LIN {X 0,Y 165.96,Z 258.398,A -85,B 0,C 180,E1 -25599.436,E2 -25599.436} C_VEL
LIN {X 0,Y 163.144,Z 293.793,A -85,B 0,C 180,E1 -25600.74,E2 -25600.74} C_VEL
LIN {X 0,Y 161.079,Z 307.116,A -85,B 0,C 180,E1 -25601.609,E2 -25601.609} C_VEL
LIN {X 0,Y 157.962,Z 319.785,A -85,B 0,C 180,E1 -25602.768,E2 -25602.768} C_VEL
LIN {X 0,Y 153.973,Z 332.432,A -85,B 0,C 180,E1 -25604.505,E2 -25604.505} C_VEL
LIN {X 0,Y 149.598,Z 343.686,A -85,B 0,C 180,E1 -25606.602,E2 -25606.602} C_VEL
LIN {X 0,Y 144.876,Z 353.82,A -85,B 0,C 180,E1 -25609.089,E2 -25609.089} C_VEL
LIN {X 0,Y 140.058,Z 362.957,A -85,B 0,C 180,E1 -25612.071,E2 -25612.071} C_VEL
LIN {X 0,Y 134.888,Z 371.867,A -85,B 0,C 180,E1 -25615.937,E2 -25615.937} C_VEL
LIN {X 0,Y 130.55,Z 379.04,A -85,B 0,C 180,E1 -25620.135,E2 -25620.135} C_VEL
LIN {X 0,Y 127.194,Z 383.879,A -85,B 0,C 180,E1 -25623.767,E2 -25623.767} C_VEL
LIN {X 0,Y 123.98,Z 388.585,A -85,B 0,C 180,E1 -25628.379,E2 -25628.379} C_VEL
LIN {X 0,Y 121.649,Z 392.184,A -85,B 0,C 180,E1 -25633.21,E2 -25633.21} C_VEL
LIN {X 0,Y 120.54,Z 394.04,A -85,B 0,C 180,E1 -25636.514,E2 -25636.514} C_VEL
LIN {X 0,Y 119.326,Z 396.429,A -85,B 0,C 180,E1 -25643.235,E2 -25643.235} C_VEL
LIN {X 0,Y 119.198,Z 397.039,A -85,B 0,C 180,E1 -25646.62,E2 -25646.62} C_VEL
LIN {X 0,Y 119.291,Z 397.251,A -85,B 0,C 180,E1 -25650,E2 -25650} C_VEL
LIN {X 0,Y 119.219,Z 397.022,A -85,B 0,C 180,E1 -25653.38,E2 -25653.38} C_VEL
LIN {X 0,Y 119.788,Z 395.395,A -85,B 0,C 180,E1 -25660.138,E2 -25660.138} C_VEL
LIN {X 0,Y 120.54,Z 393.984,A -85,B 0,C 180,E1 -25663.487,E2 -25663.487} C_VEL
LIN {X 0,Y 122.284,Z 391.031,A -85,B 0,C 180,E1 -25668.427,E2 -25668.427} C_VEL
LIN {X 0,Y 124.982,Z 387.046,A -85,B 0,C 180,E1 -25673.18,E2 -25673.18} C_VEL
LIN {X 0,Y 129.119,Z 380.92,A -85,B 0,C 180,E1 -25678.442,E2 -25678.442} C_VEL
LIN {X 0,Y 130.23,Z 379.284,A -85,B 0,C 180,E1 -25679.585,E2 -25679.585} C_VEL
LIN {X 0,Y 131.603,Z 376.213,A -85,B 0,C 180,E1 -25681.706,E2 -25681.706} C_VEL
LIN {X 0,Y 132.464,Z 370.828,A -85,B 0,C 180,E1 -25685.303,E2 -25685.303} C_VEL
LIN {X 0,Y 133.645,Z 364.946,A -85,B 0,C 180,E1 -25688.681,E2 -25688.681} C_VEL
LIN {X 0,Y 135.434,Z 360.956,A -85,B 0,C 180,E1 -25690.384,E2 -25690.384} C_VEL
LIN {X 0,Y 140.658,Z 351.229,A -85,B 0,C 180,E1 -25693.395,E2 -25693.395} C_VEL
LIN {X 0,Y 145.589,Z 340.541,A -85,B 0,C 180,E1 -25695.894,E2 -25695.894} C_VEL
LIN {X 0,Y 149.649,Z 330.202,A -85,B 0,C 180,E1 -25697.703,E2 -25697.703} C_VEL
LIN {X 0,Y 153.56,Z 317.82,A -85,B 0,C 180,E1 -25699.289,E2 -25699.289} C_VEL
LIN {X 0,Y 156.62,Z 304.973,A -85,B 0,C 180,E1 -25700.433,E2 -25700.433} C_VEL
LIN {X 0,Y 158.651,Z 292.264,A -85,B 0,C 180,E1 -25701.174,E2 -25701.174} C_VEL
LIN {X 0,Y 161.154,Z 260.477,A -85,B 0,C 180,E1 -25702.371,E2 -25702.371} C_VEL
LIN {X 0,Y 157.378,Z 250.162,A -85,B 0,C 180,E1 -25704.971,E2 -25704.971} C_VEL
LIN {X 0,Y 153.31,Z 240.715,A -85,B 0,C 180,E1 -25707.991,E2 -25707.991} C_VEL
LIN {X 0,Y 150.402,Z 235.01,A -85,B 0,C 180,E1 -25710.329,E2 -25710.329} C_VEL
LIN {X 0,Y 146.424,Z 228.751,A -85,B 0,C 180,E1 -25713.834,E2 -25713.834} C_VEL
LIN {X 0,Y 143.553,Z 224.641,A -85,B 0,C 180,E1 -25716.752,E2 -25716.752} C_VEL
LIN {X 0,Y 140.491,Z 220.322,A -85,B 0,C 180,E1 -25720.456,E2 -25720.456} C_VEL
LIN {X 0,Y 137.899,Z 216.949,A -85,B 0,C 180,E1 -25724.339,E2 -25724.339} C_VEL
LIN {X 0,Y 137.281,Z 215.591,A -85,B 0,C 180,E1 -25725.548,E2 -25725.548} C_VEL
LIN {X 0,Y 134.605,Z 212.975,A -85,B 0,C 180,E1 -25731.745,E2 -25731.745} C_VEL
LIN {X 0,Y 133.72,Z 210.009,A -85,B 0,C 180,E1 -25736.987,E2 -25736.987} C_VEL
LIN {X 0,Y 133.537,Z 209.824,A -85,B 0,C 180,E1 -25740.492,E2 -25740.492} C_VEL
LIN {X 0,Y 133.763,Z 210.322,A -85,B 0,C 180,E1 -25743.954,E2 -25743.954} C_VEL
LIN {X 0,Y 135.664,Z 214.412,A -85,B 0,C 180,E1 -25751.618,E2 -25751.618} C_VEL
LIN {X 0,Y 137.421,Z 215.89,A -85,B 0,C 180,E1 -25755.1,E2 -25755.1} C_VEL
LIN {X 0,Y 139.595,Z 219.458,A -85,B 0,C 180,E1 -25758.721,E2 -25758.721} C_VEL
LIN {X 0,Y 141.048,Z 221.001,A -85,B 0,C 180,E1 -25760.63,E2 -25760.63} C_VEL
LIN {X 0,Y 143.568,Z 224.638,A -85,B 0,C 180,E1 -25763.628,E2 -25763.628} C_VEL
LIN {X 0,Y 147.498,Z 230.419,A -85,B 0,C 180,E1 -25767.537,E2 -25767.537} C_VEL
LIN {X 0,Y 151.284,Z 236.282,A -85,B 0,C 180,E1 -25770.732,E2 -25770.732} C_VEL
LIN {X 0,Y 156.65,Z 245.798,A -85,B 0,C 180,E1 -25774.672,E2 -25774.672} C_VEL
LIN {X 0,Y 161.08,Z 254.69,A -85,B 0,C 180,E1 -25777.547,E2 -25777.547} C_VEL
LIN {X 0,Y 161.478,Z 255.745,A -85,B 0,C 180,E1 -25777.807,E2 -25777.807} C_VEL
LIN {X 0,Y 159.341,Z 283.576,A -85,B 0,C 180,E1 -25778.829,E2 -25778.829} C_VEL
LIN {X 0,Y 157.621,Z 297.006,A -85,B 0,C 180,E1 -25779.541,E2 -25779.541} C_VEL
LIN {X 0,Y 155.295,Z 308.347,A -85,B 0,C 180,E1 -25780.46,E2 -25780.46} C_VEL
LIN {X 0,Y 152.099,Z 320.167,A -85,B 0,C 180,E1 -25781.834,E2 -25781.834} C_VEL
LIN {X 0,Y 148.163,Z 331.584,A -85,B 0,C 180,E1 -25783.666,E2 -25783.666} C_VEL
LIN {X 0,Y 143.735,Z 341.971,A -85,B 0,C 180,E1 -25785.832,E2 -25785.832} C_VEL
LIN {X 0,Y 138.516,Z 352.453,A -85,B 0,C 180,E1 -25788.731,E2 -25788.731} C_VEL
LIN {X 0,Y 133.346,Z 361.706,A -85,B 0,C 180,E1 -25792.24,E2 -25792.24} C_VEL
LIN {X 0,Y 127.819,Z 370.401,A -85,B 0,C 180,E1 -25796.644,E2 -25796.644} C_VEL
LIN {X 0,Y 123.308,Z 376.812,A -85,B 0,C 180,E1 -25801.023,E2 -25801.023} C_VEL
LIN {X 0,Y 119.476,Z 381.898,A -85,B 0,C 180,E1 -25805.684,E2 -25805.684} C_VEL
LIN {X 0,Y 116.506,Z 385.843,A -85,B 0,C 180,E1 -25810.623,E2 -25810.623} C_VEL
LIN {X 0,Y 114.383,Z 388.753,A -85,B 0,C 180,E1 -25815.773,E2 -25815.773} C_VEL
LIN {X 0,Y 113.362,Z 390.143,A -85,B 0,C 180,E1 -25819.281,E2 -25819.281} C_VEL
LIN {X 0,Y 112.716,Z 391.13,A -85,B 0,C 180,E1 -25822.836,E2 -25822.836} C_VEL
LIN {X 0,Y 112.357,Z 391.736,A -85,B 0,C 180,E1 -25826.414,E2 -25826.414} C_VEL
LIN {X 0,Y 112.266,Z 391.961,A -85,B 0,C 180,E1 -25830,E2 -25830} C_VEL
LIN {X 0,Y 112.357,Z 391.765,A -85,B 0,C 180,E1 -25833.586,E2 -25833.586} C_VEL
LIN {X 0,Y 112.714,Z 391.178,A -85,B 0,C 180,E1 -25837.164,E2 -25837.164} C_VEL
LIN {X 0,Y 114.316,Z 388.851,A -85,B 0,C 180,E1 -25844.236,E2 -25844.236} C_VEL
LIN {X 0,Y 116.481,Z 385.977,A -85,B 0,C 180,E1 -25849.381,E2 -25849.381} C_VEL
LIN {X 0,Y 119.429,Z 382.078,A -85,B 0,C 180,E1 -25854.326,E2 -25854.326} C_VEL
LIN {X 0,Y 123.252,Z 377.046,A -85,B 0,C 180,E1 -25858.991,E2 -25858.991} C_VEL
LIN {X 0,Y 127.779,Z 370.705,A -85,B 0,C 180,E1 -25863.368,E2 -25863.368} C_VEL
LIN {X 0,Y 132.378,Z 363.417,A -85,B 0,C 180,E1 -25867.216,E2 -25867.216} C_VEL
LIN {X 0,Y 137.465,Z 354.696,A -85,B 0,C 180,E1 -25870.681,E2 -25870.681} C_VEL
LIN {X 0,Y 142.569,Z 344.828,A -85,B 0,C 180,E1 -25873.64,E2 -25873.64} C_VEL
LIN {X 0,Y 147.491,Z 333.709,A -85,B 0,C 180,E1 -25876.113,E2 -25876.113} C_VEL
LIN {X 0,Y 151.476,Z 322.81,A -85,B 0,C 180,E1 -25877.932,E2 -25877.932} C_VEL
LIN {X 0,Y 154.93,Z 310.758,A -85,B 0,C 180,E1 -25879.448,E2 -25879.448} C_VEL
LIN {X 0,Y 157.633,Z 297.96,A -85,B 0,C 180,E1 -25880.571,E2 -25880.571} C_VEL
LIN {X 0,Y 159.48,Z 284.567,A -85,B 0,C 180,E1 -25881.274,E2 -25881.274} C_VEL
LIN {X 0,Y 161.637,Z 255.87,A -85,B 0,C 180,E1 -25882.361,E2 -25882.361} C_VEL
LIN {X 0,Y 158.953,Z 250.067,A -85,B 0,C 180,E1 -25884.077,E2 -25884.077} C_VEL
LIN {X 0,Y 154.22,Z 241.25,A -85,B 0,C 180,E1 -25887.334,E2 -25887.334} C_VEL
LIN {X 0,Y 149.944,Z 234.02,A -85,B 0,C 180,E1 -25890.682,E2 -25890.682} C_VEL
LIN {X 0,Y 146.174,Z 228.323,A -85,B 0,C 180,E1 -25894.073,E2 -25894.073} C_VEL
LIN {X 0,Y 143.742,Z 224.785,A -85,B 0,C 180,E1 -25896.592,E2 -25896.592} C_VEL
LIN {X 0,Y 140.574,Z 220.326,A -85,B 0,C 180,E1 -25900.467,E2 -25900.467} C_VEL
LIN {X 0,Y 138.098,Z 217.177,A -85,B 0,C 180,E1 -25904.219,E2 -25904.219} C_VEL
LIN {X 0,Y 137.332,Z 215.553,A -85,B 0,C 180,E1 -25905.742,E2 -25905.742} C_VEL
LIN {X 0,Y 134.875,Z 213.248,A -85,B 0,C 180,E1 -25911.573,E2 -25911.573} C_VEL
LIN {X 0,Y 133.906,Z 209.972,A -85,B 0,C 180,E1 -25918.496,E2 -25918.496} C_VEL
LIN {X 0,Y 133.95,Z 210.252,A -85,B 0,C 180,E1 -25922.255,E2 -25922.255} C_VEL
LIN {X 0,Y 135.936,Z 214.575,A -85,B 0,C 180,E1 -25931.157,E2 -25931.157} C_VEL
LIN {X 0,Y 137.467,Z 215.748,A -85,B 0,C 180,E1 -25934.243,E2 -25934.243} C_VEL
LIN {X 0,Y 139.382,Z 219.091,A -85,B 0,C 180,E1 -25937.61,E2 -25937.61} C_VEL
LIN {X 0,Y 141.133,Z 221.068,A -85,B 0,C 180,E1 -25939.999,E2 -25939.999} C_VEL
LIN {X 0,Y 143.872,Z 224.907,A -85,B 0,C 180,E1 -25943.266,E2 -25943.266} C_VEL
LIN {X 0,Y 147.676,Z 230.597,A -85,B 0,C 180,E1 -25947.07,E2 -25947.07} C_VEL
LIN {X 0,Y 151.237,Z 236.191,A -85,B 0,C 180,E1 -25950.108,E2 -25950.108} C_VEL
LIN {X 0,Y 155.273,Z 244.8,A -85,B 0,C 180,E1 -25953.287,E2 -25953.287} C_VEL
LIN {X 0,Y 159.506,Z 255.337,A -85,B 0,C 180,E1 -25956.315,E2 -25956.315} C_VEL
LIN {X 0,Y 161.349,Z 260.706,A -85,B 0,C 180,E1 -25957.576,E2 -25957.576} C_VEL
LIN {X 0,Y 158.567,Z 293.865,A -85,B 0,C 180,E1 -25958.805,E2 -25958.805} C_VEL
LIN {X 0,Y 156.388,Z 307.31,A -85,B 0,C 180,E1 -25959.692,E2 -25959.692} C_VEL
LIN {X 0,Y 153.233,Z 319.63,A -85,B 0,C 180,E1 -25960.82,E2 -25960.82} C_VEL
LIN {X 0,Y 149.082,Z 332.275,A -85,B 0,C 180,E1 -25962.558,E2 -25962.558} C_VEL
LIN {X 0,Y 144.512,Z 343.528,A -85,B 0,C 180,E1 -25964.664,E2 -25964.664} C_VEL
LIN {X 0,Y 139.583,Z 353.661,A -85,B 0,C 180,E1 -25967.178,E2 -25967.178} C_VEL
LIN {X 0,Y 134.52,Z 362.797,A -85,B 0,C 180,E1 -25970.209,E2 -25970.209} C_VEL
LIN {X 0,Y 129.048,Z 371.707,A -85,B 0,C 180,E1 -25974.166,E2 -25974.166} C_VEL
LIN {X 0,Y 124.618,Z 378.549,A -85,B 0,C 180,E1 -25978.272,E2 -25978.272} C_VEL
LIN {X 0,Y 120.832,Z 383.717,A -85,B 0,C 180,E1 -25982.27,E2 -25982.27} C_VEL
LIN {X 0,Y 117.394,Z 388.423,A -85,B 0,C 180,E1 -25987.1,E2 -25987.1} C_VEL
LIN {X 0,Y 114.817,Z 392.021,A -85,B 0,C 180,E1 -25992.179,E2 -25992.179} C_VEL
LIN {X 0,Y 113.632,Z 393.878,A -85,B 0,C 180,E1 -25995.677,E2 -25995.677} C_VEL
LIN {X 0,Y 112.262,Z 396.267,A -85,B 0,C 180,E1 -26002.808,E2 -26002.808} C_VEL
LIN {X 0,Y 112.113,Z 396.877,A -85,B 0,C 180,E1 -26006.406,E2 -26006.406} C_VEL
LIN {X 0,Y 112.203,Z 397.09,A -85,B 0,C 180,E1 -26010,E2 -26010} C_VEL
LIN {X 0,Y 112.126,Z 396.86,A -85,B 0,C 180,E1 -26013.594,E2 -26013.594} C_VEL
LIN {X 0,Y 112.781,Z 395.232,A -85,B 0,C 180,E1 -26020.775,E2 -26020.775} C_VEL
LIN {X 0,Y 113.632,Z 393.821,A -85,B 0,C 180,E1 -26024.323,E2 -26024.323} C_VEL
LIN {X 0,Y 115.533,Z 390.867,A -85,B 0,C 180,E1 -26029.547,E2 -26029.547} C_VEL
LIN {X 0,Y 118.471,Z 386.882,A -85,B 0,C 180,E1 -26034.536,E2 -26034.536} C_VEL
LIN {X 0,Y 122.924,Z 380.756,A -85,B 0,C 180,E1 -26040.018,E2 -26040.018} C_VEL
LIN {X 0,Y 127.336,Z 374.065,A -85,B 0,C 180,E1 -26044.453,E2 -26044.453} C_VEL
LIN {X 0,Y 132.576,Z 365.773,A -85,B 0,C 180,E1 -26048.527,E2 -26048.527} C_VEL
LIN {X 0,Y 135.434,Z 360.956,A -85,B 0,C 180,E1 -26050.384,E2 -26050.384} C_VEL
LIN {X 0,Y 137.291,Z 356.824,A -85,B 0,C 180,E1 -26051.978,E2 -26051.978} C_VEL
LIN {X 0,Y 138.917,Z 349.782,A -85,B 0,C 180,E1 -26054.794,E2 -26054.794} C_VEL
LIN {X 0,Y 140.44,Z 342.254,A -85,B 0,C 180,E1 -26057.366,E2 -26057.366} C_VEL
LIN {X 0,Y 142.051,Z 337.36,A -85,B 0,C 180,E1 -26058.542,E2 -26058.542} C_VEL
LIN {X 0,Y 146.209,Z 326.549,A -85,B 0,C 180,E1 -26060.272,E2 -26060.272} C_VEL
LIN {X 0,Y 149.985,Z 314.254,A -85,B 0,C 180,E1 -26061.709,E2 -26061.709} C_VEL
LIN {X 0,Y 153.018,Z 300.61,A -85,B 0,C 180,E1 -26062.761,E2 -26062.761} C_VEL
LIN {X 0,Y 154.706,Z 288.036,A -85,B 0,C 180,E1 -26063.397,E2 -26063.397} C_VEL
LIN {X 0,Y 156.632,Z 262.443,A -85,B 0,C 180,E1 -26064.405,E2 -26064.405} C_VEL
LIN {X 0,Y 152.84,Z 252.082,A -85,B 0,C 180,E1 -26067.296,E2 -26067.296} C_VEL
LIN {X 0,Y 148.929,Z 242.938,A -85,B 0,C 180,E1 -26070.564,E2 -26070.564} C_VEL
LIN {X 0,Y 146.191,Z 238.073,A -85,B 0,C 180,E1 -26073.019,E2 -26073.019} C_VEL
LIN {X 0,Y 143.455,Z 233.842,A -85,B 0,C 180,E1 -26075.728,E2 -26075.728} C_VEL
LIN {X 0,Y 141.54,Z 230.9,A -85,B 0,C 180,E1 -26077.876,E2 -26077.876} C_VEL
LIN {X 0,Y 138.732,Z 226.775,A -85,B 0,C 180,E1 -26081.542,E2 -26081.542} C_VEL
LIN {X 0,Y 136.315,Z 223.245,A -85,B 0,C 180,E1 -26085.539,E2 -26085.539} C_VEL
LIN {X 0,Y 135.832,Z 222.322,A -85,B 0,C 180,E1 -26086.542,E2 -26086.542} C_VEL
LIN {X 0,Y 133.436,Z 219.6,A -85,B 0,C 180,E1 -26092.814,E2 -26092.814} C_VEL
LIN {X 0,Y 132.775,Z 217.004,A -85,B 0,C 180,E1 -26097.725,E2 -26097.725} C_VEL
LIN {X 0,Y 132.806,Z 217.095,A -85,B 0,C 180,E1 -26103.034,E2 -26103.034} C_VEL
LIN {X 0,Y 134.662,Z 221.446,A -85,B 0,C 180,E1 -26111.361,E2 -26111.361} C_VEL
LIN {X 0,Y 136.108,Z 222.76,A -85,B 0,C 180,E1 -26114.389,E2 -26114.389} C_VEL
LIN {X 0,Y 138.491,Z 226.554,A -85,B 0,C 180,E1 -26118.492,E2 -26118.492} C_VEL
LIN {X 0,Y 139.553,Z 227.908,A -85,B 0,C 180,E1 -26119.969,E2 -26119.969} C_VEL
LIN {X 0,Y 142.603,Z 232.443,A -85,B 0,C 180,E1 -26123.702,E2 -26123.702} C_VEL
LIN {X 0,Y 145.838,Z 237.495,A -85,B 0,C 180,E1 -26127.014,E2 -26127.014} C_VEL
LIN {X 0,Y 149.97,Z 244.505,A -85,B 0,C 180,E1 -26130.64,E2 -26130.64} C_VEL
LIN {X 0,Y 154.265,Z 252.615,A -85,B 0,C 180,E1 -26133.924,E2 -26133.924} C_VEL
LIN {X 0,Y 156.97,Z 258.26,A -85,B 0,C 180,E1 -26135.812,E2 -26135.812} C_VEL
LIN {X 0,Y 155.332,Z 280.28,A -85,B 0,C 180,E1 -26136.672,E2 -26136.672} C_VEL
LIN {X 0,Y 153.755,Z 293.786,A -85,B 0,C 180,E1 -26137.264,E2 -26137.264} C_VEL
LIN {X 0,Y 151.366,Z 305.921,A -85,B 0,C 180,E1 -26138.148,E2 -26138.148} C_VEL
LIN {X 0,Y 148.084,Z 318.374,A -85,B 0,C 180,E1 -26139.537,E2 -26139.537} C_VEL
LIN {X 0,Y 143.935,Z 330.319,A -85,B 0,C 180,E1 -26141.347,E2 -26141.347} C_VEL
LIN {X 0,Y 139.301,Z 340.966,A -85,B 0,C 180,E1 -26143.511,E2 -26143.511} C_VEL
LIN {X 0,Y 134.327,Z 350.673,A -85,B 0,C 180,E1 -26146.113,E2 -26146.113} C_VEL
LIN {X 0,Y 129.235,Z 359.503,A -85,B 0,C 180,E1 -26149.264,E2 -26149.264} C_VEL
LIN {X 0,Y 124.58,Z 366.785,A -85,B 0,C 180,E1 -26152.667,E2 -26152.667} C_VEL
LIN {X 0,Y 119.469,Z 373.952,A -85,B 0,C 180,E1 -26157.033,E2 -26157.033} C_VEL
LIN {X 0,Y 115.657,Z 378.785,A -85,B 0,C 180,E1 -26160.914,E2 -26160.914} C_VEL
LIN {X 0,Y 111.911,Z 383.477,A -85,B 0,C 180,E1 -26165.908,E2 -26165.908} C_VEL
LIN {X 0,Y 108.947,Z 387.066,A -85,B 0,C 180,E1 -26171.183,E2 -26171.183} C_VEL
LIN {X 0,Y 107.497,Z 388.916,A -85,B 0,C 180,E1 -26174.84,E2 -26174.84} C_VEL
LIN {X 0,Y 106.399,Z 390.305,A -85,B 0,C 180,E1 -26178.571,E2 -26178.571} C_VEL
LIN {X 0,Y 105.271,Z 391.898,A -85,B 0,C 180,E1 -26186.172,E2 -26186.172} C_VEL
LIN {X 0,Y 105.18,Z 392.123,A -85,B 0,C 180,E1 -26190,E2 -26190} C_VEL
LIN {X 0,Y 105.271,Z 391.927,A -85,B 0,C 180,E1 -26193.828,E2 -26193.828} C_VEL
LIN {X 0,Y 105.664,Z 391.34,A -85,B 0,C 180,E1 -26197.644,E2 -26197.644} C_VEL
LIN {X 0,Y 106.384,Z 390.372,A -85,B 0,C 180,E1 -26201.431,E2 -26201.431} C_VEL
LIN {X 0,Y 107.442,Z 389.013,A -85,B 0,C 180,E1 -26205.168,E2 -26205.168} C_VEL
LIN {X 0,Y 109.814,Z 386.138,A -85,B 0,C 180,E1 -26210.609,E2 -26210.609} C_VEL
LIN {X 0,Y 112.979,Z 382.24,A -85,B 0,C 180,E1 -26215.813,E2 -26215.813} C_VEL
LIN {X 0,Y 117.1,Z 377.206,A -85,B 0,C 180,E1 -26220.673,E2 -26220.673} C_VEL
LIN {X 0,Y 121.904,Z 370.866,A -85,B 0,C 180,E1 -26225.206,E2 -26225.206} C_VEL
LIN {X 0,Y 127.265,Z 362.82,A -85,B 0,C 180,E1 -26229.508,E2 -26229.508} C_VEL
LIN {X 0,Y 133.209,Z 353.076,A -85,B 0,C 180,E1 -26233.304,E2 -26233.304} C_VEL
LIN {X 0,Y 138.66,Z 342.71,A -85,B 0,C 180,E1 -26236.241,E2 -26236.241} C_VEL
LIN {X 0,Y 143.847,Z 331.02,A -85,B 0,C 180,E1 -26238.693,E2 -26238.693} C_VEL
LIN {X 0,Y 148.044,Z 319.342,A -85,B 0,C 180,E1 -26240.482,E2 -26240.482} C_VEL
LIN {X 0,Y 151.295,Z 307.194,A -85,B 0,C 180,E1 -26241.886,E2 -26241.886} C_VEL
LIN {X 0,Y 153.935,Z 293.999,A -85,B 0,C 180,E1 -26242.88,E2 -26242.88} C_VEL
LIN {X 0,Y 155.519,Z 280.651,A -85,B 0,C 180,E1 -26243.47,E2 -26243.47} C_VEL
LIN {X 0,Y 157.275,Z 258.655,A -85,B 0,C 180,E1 -26244.269,E2 -26244.269} C_VEL
LIN {X 0,Y 152.83,Z 249.559,A -85,B 0,C 180,E1 -26247.44,E2 -26247.44} C_VEL
LIN {X 0,Y 148.312,Z 241.396,A -85,B 0,C 180,E1 -26251.096,E2 -26251.096} C_VEL
LIN {X 0,Y 144.336,Z 234.914,A -85,B 0,C 180,E1 -26254.855,E2 -26254.855} C_VEL
LIN {X 0,Y 141.761,Z 231.044,A -85,B 0,C 180,E1 -26257.693,E2 -26257.693} C_VEL
LIN {X 0,Y 138.954,Z 226.916,A -85,B 0,C 180,E1 -26261.381,E2 -26261.381} C_VEL
LIN {X 0,Y 136.588,Z 223.641,A -85,B 0,C 180,E1 -26265.282,E2 -26265.282} C_VEL
LIN {X 0,Y 135.998,Z 222.375,A -85,B 0,C 180,E1 -26266.553,E2 -26266.553} C_VEL
LIN {X 0,Y 133.667,Z 219.806,A -85,B 0,C 180,E1 -26272.826,E2 -26272.826} C_VEL
LIN {X 0,Y 133.038,Z 217.046,A -85,B 0,C 180,E1 -26278.486,E2 -26278.486} C_VEL
LIN {X 0,Y 133.047,Z 217.217,A -85,B 0,C 180,E1 -26281.703,E2 -26281.703} C_VEL
LIN {X 0,Y 135.408,Z 222.014,A -85,B 0,C 180,E1 -26291.982,E2 -26291.982} C_VEL
LIN {X 0,Y 136.25,Z 222.814,A -85,B 0,C 180,E1 -26293.707,E2 -26293.707} C_VEL
LIN {X 0,Y 138.168,Z 226.066,A -85,B 0,C 180,E1 -26297.197,E2 -26297.197} C_VEL
LIN {X 0,Y 139.493,Z 227.71,A -85,B 0,C 180,E1 -26299.116,E2 -26299.116} C_VEL
LIN {X 0,Y 142.844,Z 232.686,A -85,B 0,C 180,E1 -26303.278,E2 -26303.278} C_VEL
LIN {X 0,Y 145.589,Z 237.012,A -85,B 0,C 180,E1 -26306.135,E2 -26306.135} C_VEL
LIN {X 0,Y 148.459,Z 241.721,A -85,B 0,C 180,E1 -26308.762,E2 -26308.762} C_VEL
LIN {X 0,Y 152.15,Z 250.015,A -85,B 0,C 180,E1 -26311.918,E2 -26311.918} C_VEL
LIN {X 0,Y 156.09,Z 260.463,A -85,B 0,C 180,E1 -26314.985,E2 -26314.985} C_VEL
LIN {X 0,Y 156.918,Z 263.011,A -85,B 0,C 180,E1 -26315.608,E2 -26315.608} C_VEL
LIN {X 0,Y 154.227,Z 293.717,A -85,B 0,C 180,E1 -26316.754,E2 -26316.754} C_VEL
LIN {X 0,Y 151.872,Z 307.507,A -85,B 0,C 180,E1 -26317.655,E2 -26317.655} C_VEL
LIN {X 0,Y 148.693,Z 319.474,A -85,B 0,C 180,E1 -26318.751,E2 -26318.751} C_VEL
LIN {X 0,Y 144.384,Z 332.118,A -85,B 0,C 180,E1 -26320.487,E2 -26320.487} C_VEL
LIN {X 0,Y 139.603,Z 343.369,A -85,B 0,C 180,E1 -26322.586,E2 -26322.586} C_VEL
LIN {X 0,Y 134.469,Z 353.502,A -85,B 0,C 180,E1 -26325.124,E2 -26325.124} C_VEL
LIN {X 0,Y 129.138,Z 362.637,A -85,B 0,C 180,E1 -26328.19,E2 -26328.19} C_VEL
LIN {X 0,Y 123.325,Z 371.545,A -85,B 0,C 180,E1 -26332.221,E2 -26332.221} C_VEL
LIN {X 0,Y 118.43,Z 378.639,A -85,B 0,C 180,E1 -26336.633,E2 -26336.633} C_VEL
LIN {X 0,Y 114.572,Z 383.556,A -85,B 0,C 180,E1 -26340.612,E2 -26340.612} C_VEL
LIN {X 0,Y 110.877,Z 388.262,A -85,B 0,C 180,E1 -26345.669,E2 -26345.669} C_VEL
LIN {X 0,Y 108.03,Z 391.859,A -85,B 0,C 180,E1 -26351.018,E2 -26351.018} C_VEL
LIN {X 0,Y 106.74,Z 393.716,A -85,B 0,C 180,E1 -26354.73,E2 -26354.73} C_VEL
LIN {X 0,Y 105.222,Z 396.105,A -85,B 0,C 180,E1 -26362.323,E2 -26362.323} C_VEL
LIN {X 0,Y 105.026,Z 396.715,A -85,B 0,C 180,E1 -26366.163,E2 -26366.163} C_VEL
LIN {X 0,Y 105.108,Z 396.927,A -85,B 0,C 180,E1 -26370,E2 -26370} C_VEL
LIN {X 0,Y 105.035,Z 396.697,A -85,B 0,C 180,E1 -26373.837,E2 -26373.837} C_VEL
LIN {X 0,Y 105.802,Z 395.069,A -85,B 0,C 180,E1 -26381.495,E2 -26381.495} C_VEL
LIN {X 0,Y 106.74,Z 393.658,A -85,B 0,C 180,E1 -26385.27,E2 -26385.27} C_VEL
LIN {X 0,Y 108.841,Z 390.704,A -85,B 0,C 180,E1 -26390.802,E2 -26390.802} C_VEL
LIN {X 0,Y 112.036,Z 386.718,A -85,B 0,C 180,E1 -26396.047,E2 -26396.047} C_VEL
LIN {X 0,Y 116.827,Z 380.592,A -85,B 0,C 180,E1 -26401.761,E2 -26401.761} C_VEL
LIN {X 0,Y 121.514,Z 373.9,A -85,B 0,C 180,E1 -26406.358,E2 -26406.358} C_VEL
LIN {X 0,Y 127.093,Z 365.608,A -85,B 0,C 180,E1 -26410.523,E2 -26410.523} C_VEL
LIN {X 0,Y 132.259,Z 357.101,A -85,B 0,C 180,E1 -26413.693,E2 -26413.693} C_VEL
LIN {X 0,Y 137.838,Z 346.593,A -85,B 0,C 180,E1 -26416.599,E2 -26416.599} C_VEL
LIN {X 0,Y 142.051,Z 337.36,A -85,B 0,C 180,E1 -26418.542,E2 -26418.542} C_VEL
LIN {X 0,Y 143.617,Z 332.355,A -85,B 0,C 180,E1 -26419.625,E2 -26419.625} C_VEL
LIN {X 0,Y 144.859,Z 323.971,A -85,B 0,C 180,E1 -26421.687,E2 -26421.687} C_VEL
LIN {X 0,Y 145.807,Z 315.311,A -85,B 0,C 180,E1 -26423.532,E2 -26423.532} C_VEL
LIN {X 0,Y 146.826,Z 309.815,A -85,B 0,C 180,E1 -26424.26,E2 -26424.26} C_VEL
LIN {X 0,Y 149.468,Z 296.815,A -85,B 0,C 180,E1 -26425.148,E2 -26425.148} C_VEL
LIN {X 0,Y 151.229,Z 280.247,A -85,B 0,C 180,E1 -26425.855,E2 -26425.855} C_VEL
LIN {X 0,Y 152.455,Z 265.218,A -85,B 0,C 180,E1 -26426.414,E2 -26426.414} C_VEL
LIN {X 0,Y 149.278,Z 256.112,A -85,B 0,C 180,E1 -26429.105,E2 -26429.105} C_VEL
LIN {X 0,Y 145.853,Z 247.69,A -85,B 0,C 180,E1 -26432.271,E2 -26432.271} C_VEL
LIN {X 0,Y 143.197,Z 243,A -85,B 0,C 180,E1 -26434.882,E2 -26434.882} C_VEL
LIN {X 0,Y 139.784,Z 237.406,A -85,B 0,C 180,E1 -26438.785,E2 -26438.785} C_VEL
LIN {X 0,Y 137.091,Z 233.299,A -85,B 0,C 180,E1 -26442.553,E2 -26442.553} C_VEL
LIN {X 0,Y 134.875,Z 229.762,A -85,B 0,C 180,E1 -26446.572,E2 -26446.572} C_VEL
LIN {X 0,Y 134.25,Z 228.973,A -85,B 0,C 180,E1 -26447.913,E2 -26447.913} C_VEL
LIN {X 0,Y 131.975,Z 224.903,A -85,B 0,C 180,E1 -26456.374,E2 -26456.374} C_VEL
LIN {X 0,Y 131.906,Z 224.089,A -85,B 0,C 180,E1 -26457.71,E2 -26457.71} C_VEL
LIN {X 0,Y 131.906,Z 224.106,A -85,B 0,C 180,E1 -26462.672,E2 -26462.672} C_VEL
LIN {X 0,Y 133.536,Z 228.308,A -85,B 0,C 180,E1 -26470.765,E2 -26470.765} C_VEL
LIN {X 0,Y 134.778,Z 229.528,A -85,B 0,C 180,E1 -26473.571,E2 -26473.571} C_VEL
LIN {X 0,Y 137.151,Z 233.383,A -85,B 0,C 180,E1 -26477.906,E2 -26477.906} C_VEL
LIN {X 0,Y 138.394,Z 235.379,A -85,B 0,C 180,E1 -26479.757,E2 -26479.757} C_VEL
LIN {X 0,Y 140.67,Z 238.82,A -85,B 0,C 180,E1 -26482.67,E2 -26482.67} C_VEL
LIN {X 0,Y 143.986,Z 244.255,A -85,B 0,C 180,E1 -26486.28,E2 -26486.28} C_VEL
LIN {X 0,Y 147.825,Z 251.238,A -85,B 0,C 180,E1 -26489.849,E2 -26489.849} C_VEL
LIN {X 0,Y 152.08,Z 259.813,A -85,B 0,C 180,E1 -26493.286,E2 -26493.286} C_VEL
LIN {X 0,Y 152.731,Z 261.258,A -85,B 0,C 180,E1 -26493.779,E2 -26493.779} C_VEL
LIN {X 0,Y 151.199,Z 280.623,A -85,B 0,C 180,E1 -26494.526,E2 -26494.526} C_VEL
LIN {X 0,Y 149.487,Z 294.409,A -85,B 0,C 180,E1 -26495.129,E2 -26495.129} C_VEL
LIN {X 0,Y 146.79,Z 307.389,A -85,B 0,C 180,E1 -26496.105,E2 -26496.105} C_VEL
LIN {X 0,Y 143.681,Z 318.542,A -85,B 0,C 180,E1 -26497.359,E2 -26497.359} C_VEL
LIN {X 0,Y 139.357,Z 330.486,A -85,B 0,C 180,E1 -26499.16,E2 -26499.16} C_VEL
LIN {X 0,Y 134.512,Z 341.132,A -85,B 0,C 180,E1 -26501.317,E2 -26501.317} C_VEL
LIN {X 0,Y 129.315,Z 350.838,A -85,B 0,C 180,E1 -26503.936,E2 -26503.936} C_VEL
LIN {X 0,Y 123.938,Z 359.668,A -85,B 0,C 180,E1 -26507.12,E2 -26507.12} C_VEL
LIN {X 0,Y 119.016,Z 366.949,A -85,B 0,C 180,E1 -26510.595,E2 -26510.595} C_VEL
LIN {X 0,Y 113.585,Z 374.116,A -85,B 0,C 180,E1 -26515.087,E2 -26515.087} C_VEL
LIN {X 0,Y 109.517,Z 378.948,A -85,B 0,C 180,E1 -26519.111,E2 -26519.111} C_VEL
LIN {X 0,Y 105.446,Z 383.641,A -85,B 0,C 180,E1 -26524.327,E2 -26524.327} C_VEL
LIN {X 0,Y 102.251,Z 387.229,A -85,B 0,C 180,E1 -26529.9,E2 -26529.9} C_VEL
LIN {X 0,Y 100.655,Z 389.079,A -85,B 0,C 180,E1 -26533.782,E2 -26533.782} C_VEL
LIN {X 0,Y 99.444,Z 390.468,A -85,B 0,C 180,E1 -26537.759,E2 -26537.759} C_VEL
LIN {X 0,Y 98.645,Z 391.455,A -85,B 0,C 180,E1 -26541.808,E2 -26541.808} C_VEL
LIN {X 0,Y 98.194,Z 392.06,A -85,B 0,C 180,E1 -26545.896,E2 -26545.896} C_VEL
LIN {X 0,Y 98.086,Z 392.285,A -85,B 0,C 180,E1 -26550,E2 -26550} C_VEL
LIN {X 0,Y 98.194,Z 392.089,A -85,B 0,C 180,E1 -26554.104,E2 -26554.104} C_VEL
LIN {X 0,Y 98.643,Z 391.502,A -85,B 0,C 180,E1 -26558.192,E2 -26558.192} C_VEL
LIN {X 0,Y 100.61,Z 389.174,A -85,B 0,C 180,E1 -26566.225,E2 -26566.225} C_VEL
LIN {X 0,Y 103.189,Z 386.3,A -85,B 0,C 180,E1 -26571.999,E2 -26571.999} C_VEL
LIN {X 0,Y 106.617,Z 382.401,A -85,B 0,C 180,E1 -26577.479,E2 -26577.479} C_VEL
LIN {X 0,Y 111.049,Z 377.367,A -85,B 0,C 180,E1 -26582.543,E2 -26582.543} C_VEL
LIN {X 0,Y 116.166,Z 371.026,A -85,B 0,C 180,E1 -26587.228,E2 -26587.228} C_VEL
LIN {X 0,Y 121.781,Z 363.103,A -85,B 0,C 180,E1 -26591.578,E2 -26591.578} C_VEL
LIN {X 0,Y 128.132,Z 353.235,A -85,B 0,C 180,E1 -26595.483,E2 -26595.483} C_VEL
LIN {X 0,Y 133.849,Z 342.868,A -85,B 0,C 180,E1 -26598.436,E2 -26598.436} C_VEL
LIN {X 0,Y 139.271,Z 331.178,A -85,B 0,C 180,E1 -26600.883,E2 -26600.883} C_VEL
LIN {X 0,Y 143.644,Z 319.497,A -85,B 0,C 180,E1 -26602.66,E2 -26602.66} C_VEL
LIN {X 0,Y 147.025,Z 307.347,A -85,B 0,C 180,E1 -26604.06,E2 -26604.06} C_VEL
LIN {X 0,Y 149.785,Z 294.014,A -85,B 0,C 180,E1 -26605.053,E2 -26605.053} C_VEL
LIN {X 0,Y 151.512,Z 279.601,A -85,B 0,C 180,E1 -26605.666,E2 -26605.666} C_VEL
LIN {X 0,Y 152.995,Z 261.546,A -85,B 0,C 180,E1 -26606.332,E2 -26606.332} C_VEL
LIN {X 0,Y 148.495,Z 252.312,A -85,B 0,C 180,E1 -26609.915,E2 -26609.915} C_VEL
LIN {X 0,Y 144.458,Z 244.763,A -85,B 0,C 180,E1 -26613.644,E2 -26613.644} C_VEL
LIN {X 0,Y 141.075,Z 239.3,A -85,B 0,C 180,E1 -26617.289,E2 -26617.289} C_VEL
LIN {X 0,Y 139.691,Z 237.181,A -85,B 0,C 180,E1 -26618.994,E2 -26618.994} C_VEL
LIN {X 0,Y 137.37,Z 233.506,A -85,B 0,C 180,E1 -26622.316,E2 -26622.316} C_VEL
LIN {X 0,Y 135.009,Z 229.81,A -85,B 0,C 180,E1 -26626.644,E2 -26626.644} C_VEL
LIN {X 0,Y 134.6,Z 229.175,A -85,B 0,C 180,E1 -26627.562,E2 -26627.562} C_VEL
LIN {X 0,Y 132.152,Z 224.537,A -85,B 0,C 180,E1 -26637.966,E2 -26637.966} C_VEL
LIN {X 0,Y 132.158,Z 224.074,A -85,B 0,C 180,E1 -26638.838,E2 -26638.838} C_VEL
LIN {X 0,Y 132.156,Z 224.38,A -85,B 0,C 180,E1 -26641.542,E2 -26641.542} C_VEL
LIN {X 0,Y 134.555,Z 229.119,A -85,B 0,C 180,E1 -26652.059,E2 -26652.059} C_VEL
LIN {X 0,Y 135.046,Z 229.874,A -85,B 0,C 180,E1 -26653.161,E2 -26653.161} C_VEL
LIN {X 0,Y 137.305,Z 233.422,A -85,B 0,C 180,E1 -26657.308,E2 -26657.308} C_VEL
LIN {X 0,Y 140.787,Z 238.782,A -85,B 0,C 180,E1 -26662.083,E2 -26662.083} C_VEL
LIN {X 0,Y 144.52,Z 244.944,A -85,B 0,C 180,E1 -26666.149,E2 -26666.149} C_VEL
LIN {X 0,Y 146.755,Z 249.444,A -85,B 0,C 180,E1 -26668.32,E2 -26668.32} C_VEL
LIN {X 0,Y 150.218,Z 258.234,A -85,B 0,C 180,E1 -26671.463,E2 -26671.463} C_VEL
LIN {X 0,Y 152.678,Z 265.36,A -85,B 0,C 180,E1 -26673.53,E2 -26673.53} C_VEL
LIN {X 0,Y 150.094,Z 293.516,A -85,B 0,C 180,E1 -26674.579,E2 -26674.579} C_VEL
LIN {X 0,Y 147.659,Z 307.266,A -85,B 0,C 180,E1 -26675.465,E2 -26675.465} C_VEL
LIN {X 0,Y 144.359,Z 319.318,A -85,B 0,C 180,E1 -26676.555,E2 -26676.555} C_VEL
LIN {X 0,Y 139.88,Z 331.961,A -85,B 0,C 180,E1 -26678.276,E2 -26678.276} C_VEL
LIN {X 0,Y 134.908,Z 343.212,A -85,B 0,C 180,E1 -26680.37,E2 -26680.37} C_VEL
LIN {X 0,Y 129.544,Z 353.343,A -85,B 0,C 180,E1 -26682.913,E2 -26682.913} C_VEL
LIN {X 0,Y 123.914,Z 362.477,A -85,B 0,C 180,E1 -26685.991,E2 -26685.991} C_VEL
LIN {X 0,Y 117.773,Z 371.385,A -85,B 0,C 180,E1 -26690.097,E2 -26690.097} C_VEL
LIN {X 0,Y 113.052,Z 377.79,A -85,B 0,C 180,E1 -26694.143,E2 -26694.143} C_VEL
LIN {X 0,Y 108.426,Z 383.395,A -85,B 0,C 180,E1 -26698.765,E2 -26698.765} C_VEL
LIN {X 0,Y 104.415,Z 388.1,A -85,B 0,C 180,E1 -26704.056,E2 -26704.056} C_VEL
LIN {X 0,Y 101.299,Z 391.696,A -85,B 0,C 180,E1 -26709.703,E2 -26709.703} C_VEL
LIN {X 0,Y 99.863,Z 393.553,A -85,B 0,C 180,E1 -26713.65,E2 -26713.65} C_VEL
LIN {X 0,Y 98.179,Z 395.943,A -85,B 0,C 180,E1 -26721.769,E2 -26721.769} C_VEL
LIN {X 0,Y 97.934,Z 396.552,A -85,B 0,C 180,E1 -26725.885,E2 -26725.885} C_VEL
LIN {X 0,Y 98.006,Z 396.765,A -85,B 0,C 180,E1 -26730,E2 -26730} C_VEL
LIN {X 0,Y 97.941,Z 396.534,A -85,B 0,C 180,E1 -26734.115,E2 -26734.115} C_VEL
LIN {X 0,Y 98.186,Z 395.914,A -85,B 0,C 180,E1 -26738.231,E2 -26738.231} C_VEL
LIN {X 0,Y 98.82,Z 394.905,A -85,B 0,C 180,E1 -26742.319,E2 -26742.319} C_VEL
LIN {X 0,Y 99.863,Z 393.494,A -85,B 0,C 180,E1 -26746.35,E2 -26746.35} C_VEL
LIN {X 0,Y 102.216,Z 390.54,A -85,B 0,C 180,E1 -26752.22,E2 -26752.22} C_VEL
LIN {X 0,Y 105.691,Z 386.554,A -85,B 0,C 180,E1 -26757.741,E2 -26757.741} C_VEL
LIN {X 0,Y 110.838,Z 380.428,A -85,B 0,C 180,E1 -26763.698,E2 -26763.698} C_VEL
LIN {X 0,Y 115.846,Z 373.735,A -85,B 0,C 180,E1 -26768.45,E2 -26768.45} C_VEL
LIN {X 0,Y 121.78,Z 365.443,A -85,B 0,C 180,E1 -26772.695,E2 -26772.695} C_VEL
LIN {X 0,Y 127.214,Z 356.935,A -85,B 0,C 180,E1 -26775.905,E2 -26775.905} C_VEL
LIN {X 0,Y 133.042,Z 346.427,A -85,B 0,C 180,E1 -26778.83,E2 -26778.83} C_VEL
LIN {X 0,Y 138.568,Z 334.593,A -85,B 0,C 180,E1 -26781.242,E2 -26781.242} C_VEL
LIN {X 0,Y 143.065,Z 322.656,A -85,B 0,C 180,E1 -26782.965,E2 -26782.965} C_VEL
LIN {X 0,Y 146.826,Z 309.815,A -85,B 0,C 180,E1 -26784.26,E2 -26784.26} C_VEL
LIN {X 0,Y 147.723,Z 304.216,A -85,B 0,C 180,E1 -26784.916,E2 -26784.916} C_VEL
LIN {X 0,Y 147.659,Z 295.046,A -85,B 0,C 180,E1 -26786.396,E2 -26786.396} C_VEL
LIN {X 0,Y 147.197,Z 285.737,A -85,B 0,C 180,E1 -26787.733,E2 -26787.733} C_VEL
LIN {X 0,Y 147.38,Z 279.92,A -85,B 0,C 180,E1 -26788.141,E2 -26788.141} C_VEL
LIN {X 0,Y 148.404,Z 267.688,A -85,B 0,C 180,E1 -26788.605,E2 -26788.605} C_VEL
LIN {X 0,Y 145.3,Z 258.558,A -85,B 0,C 180,E1 -26791.567,E2 -26791.567} C_VEL
LIN {X 0,Y 142.843,Z 252.411,A -85,B 0,C 180,E1 -26794.109,E2 -26794.109} C_VEL
LIN {X 0,Y 139.467,Z 246.375,A -85,B 0,C 180,E1 -26797.894,E2 -26797.894} C_VEL
LIN {X 0,Y 137.549,Z 243.184,A -85,B 0,C 180,E1 -26800.409,E2 -26800.409} C_VEL
LIN {X 0,Y 135.589,Z 239.932,A -85,B 0,C 180,E1 -26803.436,E2 -26803.436} C_VEL
LIN {X 0,Y 133.226,Z 235.965,A -85,B 0,C 180,E1 -26808.205,E2 -26808.205} C_VEL
LIN {X 0,Y 131.121,Z 232.241,A -85,B 0,C 180,E1 -26816.062,E2 -26816.062} C_VEL
LIN {X 0,Y 130.988,Z 231.049,A -85,B 0,C 180,E1 -26818.463,E2 -26818.463} C_VEL
LIN {X 0,Y 131.007,Z 231.28,A -85,B 0,C 180,E1 -26822.498,E2 -26822.498} C_VEL
LIN {X 0,Y 132.672,Z 235.476,A -85,B 0,C 180,E1 -26830.836,E2 -26830.836} C_VEL
LIN {X 0,Y 133.551,Z 236.468,A -85,B 0,C 180,E1 -26832.924,E2 -26832.924} C_VEL
LIN {X 0,Y 136.323,Z 241.051,A -85,B 0,C 180,E1 -26838.116,E2 -26838.116} C_VEL
LIN {X 0,Y 139.053,Z 245.655,A -85,B 0,C 180,E1 -26841.954,E2 -26841.954} C_VEL
LIN {X 0,Y 142.182,Z 251.079,A -85,B 0,C 180,E1 -26845.554,E2 -26845.554} C_VEL
LIN {X 0,Y 146.175,Z 258.928,A -85,B 0,C 180,E1 -26849.459,E2 -26849.459} C_VEL
LIN {X 0,Y 148.655,Z 264.308,A -85,B 0,C 180,E1 -26851.612,E2 -26851.612} C_VEL
LIN {X 0,Y 147.16,Z 282.19,A -85,B 0,C 180,E1 -26852.293,E2 -26852.293} C_VEL
LIN {X 0,Y 145.334,Z 295.692,A -85,B 0,C 180,E1 -26852.924,E2 -26852.924} C_VEL
LIN {X 0,Y 142.403,Z 308.858,A -85,B 0,C 180,E1 -26853.927,E2 -26853.927} C_VEL
LIN {X 0,Y 138.826,Z 320.671,A -85,B 0,C 180,E1 -26855.282,E2 -26855.282} C_VEL
LIN {X 0,Y 134.355,Z 332.084,A -85,B 0,C 180,E1 -26857.088,E2 -26857.088} C_VEL
LIN {X 0,Y 129.334,Z 342.468,A -85,B 0,C 180,E1 -26859.254,E2 -26859.254} C_VEL
LIN {X 0,Y 123.31,Z 352.949,A -85,B 0,C 180,E1 -26862.19,E2 -26862.19} C_VEL
LIN {X 0,Y 117.84,Z 361.325,A -85,B 0,C 180,E1 -26865.432,E2 -26865.432} C_VEL
LIN {X 0,Y 111.601,Z 369.667,A -85,B 0,C 180,E1 -26869.798,E2 -26869.798} C_VEL
LIN {X 0,Y 106.027,Z 376.308,A -85,B 0,C 180,E1 -26874.55,E2 -26874.55} C_VEL
LIN {X 0,Y 100.404,Z 382.389,A -85,B 0,C 180,E1 -26880.661,E2 -26880.661} C_VEL
LIN {X 0,Y 96.659,Z 386.332,A -85,B 0,C 180,E1 -26886.428,E2 -26886.428} C_VEL
LIN {X 0,Y 93.862,Z 389.242,A -85,B 0,C 180,E1 -26892.572,E2 -26892.572} C_VEL
LIN {X 0,Y 91.619,Z 391.618,A -85,B 0,C 180,E1 -26901.175,E2 -26901.175} C_VEL
LIN {X 0,Y 91.113,Z 392.223,A -85,B 0,C 180,E1 -26905.576,E2 -26905.576} C_VEL
LIN {X 0,Y 91.003,Z 392.447,A -85,B 0,C 180,E1 -26910,E2 -26910} C_VEL
LIN {X 0,Y 91.113,Z 392.251,A -85,B 0,C 180,E1 -26914.424,E2 -26914.424} C_VEL
LIN {X 0,Y 91.616,Z 391.664,A -85,B 0,C 180,E1 -26918.825,E2 -26918.825} C_VEL
LIN {X 0,Y 93.796,Z 389.336,A -85,B 0,C 180,E1 -26927.44,E2 -26927.44} C_VEL
LIN {X 0,Y 96.638,Z 386.461,A -85,B 0,C 180,E1 -26933.577,E2 -26933.577} C_VEL
LIN {X 0,Y 100.356,Z 382.563,A -85,B 0,C 180,E1 -26939.354,E2 -26939.354} C_VEL
LIN {X 0,Y 105.122,Z 377.528,A -85,B 0,C 180,E1 -26944.629,E2 -26944.629} C_VEL
LIN {X 0,Y 110.58,Z 371.187,A -85,B 0,C 180,E1 -26949.461,E2 -26949.461} C_VEL
LIN {X 0,Y 116.348,Z 363.556,A -85,B 0,C 180,E1 -26953.759,E2 -26953.759} C_VEL
LIN {X 0,Y 122.096,Z 355.174,A -85,B 0,C 180,E1 -26957.214,E2 -26957.214} C_VEL
LIN {X 0,Y 128.017,Z 345.304,A -85,B 0,C 180,E1 -26960.227,E2 -26960.227} C_VEL
LIN {X 0,Y 133.634,Z 334.181,A -85,B 0,C 180,E1 -26962.697,E2 -26962.697} C_VEL
LIN {X 0,Y 138.112,Z 323.279,A -85,B 0,C 180,E1 -26964.505,E2 -26964.505} C_VEL
LIN {X 0,Y 142.021,Z 311.222,A -85,B 0,C 180,E1 -26965.984,E2 -26965.984} C_VEL
LIN {X 0,Y 145.039,Z 298.558,A -85,B 0,C 180,E1 -26967.059,E2 -26967.059} C_VEL
LIN {X 0,Y 147.159,Z 284.677,A -85,B 0,C 180,E1 -26967.755,E2 -26967.755} C_VEL
LIN {X 0,Y 148.948,Z 264.717,A -85,B 0,C 180,E1 -26968.471,E2 -26968.471} C_VEL
LIN {X 0,Y 144.98,Z 256.2,A -85,B 0,C 180,E1 -26972.016,E2 -26972.016} C_VEL
LIN {X 0,Y 141.479,Z 249.671,A -85,B 0,C 180,E1 -26975.61,E2 -26975.61} C_VEL
LIN {X 0,Y 138.416,Z 244.236,A -85,B 0,C 180,E1 -26979.375,E2 -26979.375} C_VEL
LIN {X 0,Y 135.718,Z 239.93,A -85,B 0,C 180,E1 -26983.452,E2 -26983.452} C_VEL
LIN {X 0,Y 133.576,Z 236.17,A -85,B 0,C 180,E1 -26987.851,E2 -26987.851} C_VEL
LIN {X 0,Y 131.265,Z 231.457,A -85,B 0,C 180,E1 -26998.537,E2 -26998.537} C_VEL
LIN {X 0,Y 131.277,Z 231.075,A -85,B 0,C 180,E1 -27000,E2 -27000} C_VEL
LIN {X 0,Y 131.324,Z 232.368,A -85,B 0,C 180,E1 -27003.068,E2 -27003.068} C_VEL
LIN {X 0,Y 133.713,Z 236.517,A -85,B 0,C 180,E1 -27012.233,E2 -27012.233} C_VEL
LIN {X 0,Y 136.409,Z 241.067,A -85,B 0,C 180,E1 -27017.426,E2 -27017.426} C_VEL
LIN {X 0,Y 138.984,Z 245.312,A -85,B 0,C 180,E1 -27021.118,E2 -27021.118} C_VEL
LIN {X 0,Y 141.248,Z 249.301,A -85,B 0,C 180,E1 -27023.859,E2 -27023.859} C_VEL
LIN {X 0,Y 143.636,Z 253.856,A -85,B 0,C 180,E1 -27026.42,E2 -27026.42} C_VEL
LIN {X 0,Y 146.765,Z 262.212,A -85,B 0,C 180,E1 -27029.586,E2 -27029.586} C_VEL
LIN {X 0,Y 148.637,Z 267.832,A -85,B 0,C 180,E1 -27031.34,E2 -27031.34} C_VEL
LIN {X 0,Y 146.189,Z 293.287,A -85,B 0,C 180,E1 -27032.281,E2 -27032.281} C_VEL
LIN {X 0,Y 143.735,Z 306.786,A -85,B 0,C 180,E1 -27033.138,E2 -27033.138} C_VEL
LIN {X 0,Y 140.251,Z 319.163,A -85,B 0,C 180,E1 -27034.228,E2 -27034.228} C_VEL
LIN {X 0,Y 135.594,Z 331.803,A -85,B 0,C 180,E1 -27035.918,E2 -27035.918} C_VEL
LIN {X 0,Y 130.419,Z 343.053,A -85,B 0,C 180,E1 -27037.991,E2 -27037.991} C_VEL
LIN {X 0,Y 124.817,Z 353.184,A -85,B 0,C 180,E1 -27040.524,E2 -27040.524} C_VEL
LIN {X 0,Y 118.884,Z 362.316,A -85,B 0,C 180,E1 -27043.6,E2 -27043.6} C_VEL
LIN {X 0,Y 112.397,Z 371.224,A -85,B 0,C 180,E1 -27047.765,E2 -27047.765} C_VEL
LIN {X 0,Y 106.935,Z 378.147,A -85,B 0,C 180,E1 -27052.291,E2 -27052.291} C_VEL
LIN {X 0,Y 102.412,Z 383.234,A -85,B 0,C 180,E1 -27056.702,E2 -27056.702} C_VEL
LIN {X 0,Y 98.055,Z 387.938,A -85,B 0,C 180,E1 -27062.233,E2 -27062.233} C_VEL
LIN {X 0,Y 94.634,Z 391.534,A -85,B 0,C 180,E1 -27068.203,E2 -27068.203} C_VEL
LIN {X 0,Y 93.036,Z 393.39,A -85,B 0,C 180,E1 -27072.413,E2 -27072.413} C_VEL
LIN {X 0,Y 91.14,Z 395.781,A -85,B 0,C 180,E1 -27081.128,E2 -27081.128} C_VEL
LIN {X 0,Y 90.837,Z 396.39,A -85,B 0,C 180,E1 -27085.563,E2 -27085.563} C_VEL
LIN {X 0,Y 90.913,Z 396.603,A -85,B 0,C 180,E1 -27090,E2 -27090} C_VEL
LIN {X 0,Y 90.871,Z 396.372,A -85,B 0,C 180,E1 -27094.436,E2 -27094.436} C_VEL
LIN {X 0,Y 91.872,Z 394.742,A -85,B 0,C 180,E1 -27103.267,E2 -27103.267} C_VEL
LIN {X 0,Y 93.036,Z 393.33,A -85,B 0,C 180,E1 -27107.588,E2 -27107.588} C_VEL
LIN {X 0,Y 95.67,Z 390.377,A -85,B 0,C 180,E1 -27113.831,E2 -27113.831} C_VEL
LIN {X 0,Y 99.433,Z 386.39,A -85,B 0,C 180,E1 -27119.654,E2 -27119.654} C_VEL
LIN {X 0,Y 104.976,Z 380.263,A -85,B 0,C 180,E1 -27125.86,E2 -27125.86} C_VEL
LIN {X 0,Y 110.348,Z 373.57,A -85,B 0,C 180,E1 -27130.754,E2 -27130.754} C_VEL
LIN {X 0,Y 116.642,Z 365.278,A -85,B 0,C 180,E1 -27135.07,E2 -27135.07} C_VEL
LIN {X 0,Y 122.376,Z 356.77,A -85,B 0,C 180,E1 -27138.295,E2 -27138.295} C_VEL
LIN {X 0,Y 128.471,Z 346.26,A -85,B 0,C 180,E1 -27141.219,E2 -27141.219} C_VEL
LIN {X 0,Y 134.236,Z 334.427,A -85,B 0,C 180,E1 -27143.607,E2 -27143.607} C_VEL
LIN {X 0,Y 138.916,Z 322.488,A -85,B 0,C 180,E1 -27145.297,E2 -27145.297} C_VEL
LIN {X 0,Y 142.694,Z 310.055,A -85,B 0,C 180,E1 -27146.533,E2 -27146.533} C_VEL
LIN {X 0,Y 145.494,Z 296.846,A -85,B 0,C 180,E1 -27147.434,E2 -27147.434} C_VEL
LIN {X 0,Y 147.208,Z 281.892,A -85,B 0,C 180,E1 -27148.07,E2 -27148.07} C_VEL
LIN {X 0,Y 147.38,Z 279.92,A -85,B 0,C 180,E1 -27148.141,E2 -27148.141} C_VEL
LIN {X 0,Y 147.346,Z 276.798,A -85,B 0,C 180,E1 -27148.445,E2 -27148.445} C_VEL
LIN {X 0,Y 146.483,Z 272.937,A -85,B 0,C 180,E1 -27149.354,E2 -27149.354} C_VEL
LIN {X 0,Y 142.439,Z 263.614,A -85,B 0,C 180,E1 -27153.197,E2 -27153.197} C_VEL
LIN {X 0,Y 140.346,Z 257.967,A -85,B 0,C 180,E1 -27155.599,E2 -27155.599} C_VEL
LIN {X 0,Y 137.342,Z 252.264,A -85,B 0,C 180,E1 -27159.304,E2 -27159.304} C_VEL
LIN {X 0,Y 135.681,Z 249.359,A -85,B 0,C 180,E1 -27161.698,E2 -27161.698} C_VEL
LIN {X 0,Y 133.975,Z 246.345,A -85,B 0,C 180,E1 -27164.6,E2 -27164.6} C_VEL
LIN {X 0,Y 132.045,Z 242.83,A -85,B 0,C 180,E1 -27168.876,E2 -27168.876} C_VEL
LIN {X 0,Y 130.176,Z 239.12,A -85,B 0,C 180,E1 -27176.712,E2 -27176.712} C_VEL
LIN {X 0,Y 130.087,Z 238.049,A -85,B 0,C 180,E1 -27179.226,E2 -27179.226} C_VEL
LIN {X 0,Y 130.11,Z 238.331,A -85,B 0,C 180,E1 -27182.128,E2 -27182.128} C_VEL
LIN {X 0,Y 131.654,Z 242.459,A -85,B 0,C 180,E1 -27190.494,E2 -27190.494} C_VEL
LIN {X 0,Y 132.346,Z 243.38,A -85,B 0,C 180,E1 -27192.264,E2 -27192.264} C_VEL
LIN {X 0,Y 134.838,Z 247.81,A -85,B 0,C 180,E1 -27197.293,E2 -27197.293} C_VEL
LIN {X 0,Y 137.167,Z 251.938,A -85,B 0,C 180,E1 -27200.822,E2 -27200.822} C_VEL
LIN {X 0,Y 139.862,Z 256.872,A -85,B 0,C 180,E1 -27204.196,E2 -27204.196} C_VEL
LIN {X 0,Y 143.599,Z 264.727,A -85,B 0,C 180,E1 -27208.181,E2 -27208.181} C_VEL
LIN {X 0,Y 144.816,Z 267.609,A -85,B 0,C 180,E1 -27209.362,E2 -27209.362} C_VEL
LIN {X 0,Y 142.922,Z 287.519,A -85,B 0,C 180,E1 -27210.091,E2 -27210.091} C_VEL
LIN {X 0,Y 140.659,Z 300.66,A -85,B 0,C 180,E1 -27210.832,E2 -27210.832} C_VEL
LIN {X 0,Y 137.568,Z 312.569,A -85,B 0,C 180,E1 -27211.861,E2 -27211.861} C_VEL
LIN {X 0,Y 133.531,Z 324.373,A -85,B 0,C 180,E1 -27213.329,E2 -27213.329} C_VEL
LIN {X 0,Y 128.869,Z 335.097,A -85,B 0,C 180,E1 -27215.111,E2 -27215.111} C_VEL
LIN {X 0,Y 123.041,Z 346.027,A -85,B 0,C 180,E1 -27217.578,E2 -27217.578} C_VEL
LIN {X 0,Y 117.434,Z 354.916,A -85,B 0,C 180,E1 -27220.267,E2 -27220.267} C_VEL
LIN {X 0,Y 111.472,Z 363.363,A -85,B 0,C 180,E1 -27223.789,E2 -27223.789} C_VEL
LIN {X 0,Y 105.225,Z 371.058,A -85,B 0,C 180,E1 -27228.095,E2 -27228.095} C_VEL
LIN {X 0,Y 99.419,Z 377.467,A -85,B 0,C 180,E1 -27233.067,E2 -27233.067} C_VEL
LIN {X 0,Y 94.267,Z 382.553,A -85,B 0,C 180,E1 -27238.541,E2 -27238.541} C_VEL
LIN {X 0,Y 90.18,Z 386.496,A -85,B 0,C 180,E1 -27244.619,E2 -27244.619} C_VEL
LIN {X 0,Y 87.095,Z 389.405,A -85,B 0,C 180,E1 -27251.169,E2 -27251.169} C_VEL
LIN {X 0,Y 85.609,Z 390.793,A -85,B 0,C 180,E1 -27255.742,E2 -27255.742} C_VEL
LIN {X 0,Y 84.622,Z 391.78,A -85,B 0,C 180,E1 -27260.438,E2 -27260.438} C_VEL
LIN {X 0,Y 84.057,Z 392.385,A -85,B 0,C 180,E1 -27265.204,E2 -27265.204} C_VEL
LIN {X 0,Y 83.924,Z 392.609,A -85,B 0,C 180,E1 -27270,E2 -27270} C_VEL
LIN {X 0,Y 84.057,Z 392.413,A -85,B 0,C 180,E1 -27274.796,E2 -27274.796} C_VEL
LIN {X 0,Y 84.619,Z 391.826,A -85,B 0,C 180,E1 -27279.561,E2 -27279.561} C_VEL
LIN {X 0,Y 87.04,Z 389.498,A -85,B 0,C 180,E1 -27288.843,E2 -27288.843} C_VEL
LIN {X 0,Y 90.158,Z 386.623,A -85,B 0,C 180,E1 -27295.387,E2 -27295.387} C_VEL
LIN {X 0,Y 94.217,Z 382.724,A -85,B 0,C 180,E1 -27301.477,E2 -27301.477} C_VEL
LIN {X 0,Y 99.356,Z 377.689,A -85,B 0,C 180,E1 -27306.959,E2 -27306.959} C_VEL
LIN {X 0,Y 105.179,Z 371.348,A -85,B 0,C 180,E1 -27311.927,E2 -27311.927} C_VEL
LIN {X 0,Y 111.545,Z 363.423,A -85,B 0,C 180,E1 -27316.43,E2 -27316.43} C_VEL
LIN {X 0,Y 118.612,Z 353.553,A -85,B 0,C 180,E1 -27320.378,E2 -27320.378} C_VEL
LIN {X 0,Y 124.876,Z 343.185,A -85,B 0,C 180,E1 -27323.32,E2 -27323.32} C_VEL
LIN {X 0,Y 130.786,Z 331.492,A -85,B 0,C 180,E1 -27325.71,E2 -27325.71} C_VEL
LIN {X 0,Y 135.518,Z 319.808,A -85,B 0,C 180,E1 -27327.429,E2 -27327.429} C_VEL
LIN {X 0,Y 139.177,Z 307.654,A -85,B 0,C 180,E1 -27328.791,E2 -27328.791} C_VEL
LIN {X 0,Y 142.016,Z 295.027,A -85,B 0,C 180,E1 -27329.692,E2 -27329.692} C_VEL
LIN {X 0,Y 143.823,Z 281.668,A -85,B 0,C 180,E1 -27330.271,E2 -27330.271} C_VEL
LIN {X 0,Y 145.058,Z 267.807,A -85,B 0,C 180,E1 -27330.777,E2 -27330.777} C_VEL
LIN {X 0,Y 141.699,Z 260.357,A -85,B 0,C 180,E1 -27334.161,E2 -27334.161} C_VEL
LIN {X 0,Y 139.138,Z 255.294,A -85,B 0,C 180,E1 -27337.102,E2 -27337.102} C_VEL
LIN {X 0,Y 136.261,Z 250.083,A -85,B 0,C 180,E1 -27340.999,E2 -27340.999} C_VEL
LIN {X 0,Y 134.232,Z 246.526,A -85,B 0,C 180,E1 -27344.409,E2 -27344.409} C_VEL
LIN {X 0,Y 132.242,Z 242.891,A -85,B 0,C 180,E1 -27348.892,E2 -27348.892} C_VEL
LIN {X 0,Y 130.41,Z 238.139,A -85,B 0,C 180,E1 -27360,E2 -27360} C_VEL
LIN {X 0,Y 132.483,Z 243.341,A -85,B 0,C 180,E1 -27371.474,E2 -27371.474} C_VEL
LIN {X 0,Y 134.925,Z 247.754,A -85,B 0,C 180,E1 -27376.569,E2 -27376.569} C_VEL
LIN {X 0,Y 137.177,Z 251.703,A -85,B 0,C 180,E1 -27380.056,E2 -27380.056} C_VEL
LIN {X 0,Y 140.019,Z 256.958,A -85,B 0,C 180,E1 -27383.675,E2 -27383.675} C_VEL
LIN {X 0,Y 141.762,Z 261.176,A -85,B 0,C 180,E1 -27385.708,E2 -27385.708} C_VEL
LIN {X 0,Y 144.654,Z 269.911,A -85,B 0,C 180,E1 -27388.869,E2 -27388.869} C_VEL
LIN {X 0,Y 144.807,Z 270.475,A -85,B 0,C 180,E1 -27389.034,E2 -27389.034} C_VEL
LIN {X 0,Y 142.57,Z 292.896,A -85,B 0,C 180,E1 -27389.862,E2 -27389.862} C_VEL
LIN {X 0,Y 140.009,Z 306.512,A -85,B 0,C 180,E1 -27390.695,E2 -27390.695} C_VEL
LIN {X 0,Y 136.391,Z 319.007,A -85,B 0,C 180,E1 -27391.765,E2 -27391.765} C_VEL
LIN {X 0,Y 131.559,Z 331.646,A -85,B 0,C 180,E1 -27393.416,E2 -27393.416} C_VEL
LIN {X 0,Y 126.168,Z 342.895,A -85,B 0,C 180,E1 -27395.447,E2 -27395.447} C_VEL
LIN {X 0,Y 120.319,Z 353.025,A -85,B 0,C 180,E1 -27397.95,E2 -27397.95} C_VEL
LIN {X 0,Y 114.087,Z 362.156,A -85,B 0,C 180,E1 -27401.008,E2 -27401.008} C_VEL
LIN {X 0,Y 107.225,Z 371.063,A -85,B 0,C 180,E1 -27405.203,E2 -27405.203} C_VEL
LIN {X 0,Y 101.756,Z 377.502,A -85,B 0,C 180,E1 -27409.441,E2 -27409.441} C_VEL
LIN {X 0,Y 96.551,Z 383.073,A -85,B 0,C 180,E1 -27414.386,E2 -27414.386} C_VEL
LIN {X 0,Y 91.812,Z 387.777,A -85,B 0,C 180,E1 -27420.162,E2 -27420.162} C_VEL
LIN {X 0,Y 88.049,Z 391.372,A -85,B 0,C 180,E1 -27426.479,E2 -27426.479} C_VEL
LIN {X 0,Y 86.266,Z 393.228,A -85,B 0,C 180,E1 -27430.982,E2 -27430.982} C_VEL
LIN {X 0,Y 84.128,Z 395.619,A -85,B 0,C 180,E1 -27440.382,E2 -27440.382} C_VEL
LIN {X 0,Y 83.762,Z 396.228,A -85,B 0,C 180,E1 -27445.187,E2 -27445.187} C_VEL
LIN {X 0,Y 83.81,Z 396.441,A -85,B 0,C 180,E1 -27450,E2 -27450} C_VEL
LIN {X 0,Y 83.787,Z 396.21,A -85,B 0,C 180,E1 -27454.812,E2 -27454.812} C_VEL
LIN {X 0,Y 84.962,Z 394.579,A -85,B 0,C 180,E1 -27464.369,E2 -27464.369} C_VEL
LIN {X 0,Y 86.267,Z 393.166,A -85,B 0,C 180,E1 -27469.019,E2 -27469.019} C_VEL
LIN {X 0,Y 89.186,Z 390.213,A -85,B 0,C 180,E1 -27475.684,E2 -27475.684} C_VEL
LIN {X 0,Y 93.29,Z 386.226,A -85,B 0,C 180,E1 -27481.826,E2 -27481.826} C_VEL
LIN {X 0,Y 99.263,Z 380.098,A -85,B 0,C 180,E1 -27488.281,E2 -27488.281} C_VEL
LIN {X 0,Y 105.045,Z 373.405,A -85,B 0,C 180,E1 -27493.297,E2 -27493.297} C_VEL
LIN {X 0,Y 111.735,Z 365.114,A -85,B 0,C 180,E1 -27497.651,E2 -27497.651} C_VEL
LIN {X 0,Y 117.774,Z 356.605,A -85,B 0,C 180,E1 -27500.874,E2 -27500.874} C_VEL
LIN {X 0,Y 124.149,Z 346.095,A -85,B 0,C 180,E1 -27503.773,E2 -27503.773} C_VEL
LIN {X 0,Y 130.149,Z 334.26,A -85,B 0,C 180,E1 -27506.124,E2 -27506.124} C_VEL
LIN {X 0,Y 135.01,Z 322.32,A -85,B 0,C 180,E1 -27507.768,E2 -27507.768} C_VEL
LIN {X 0,Y 138.904,Z 309.885,A -85,B 0,C 180,E1 -27508.978,E2 -27508.978} C_VEL
LIN {X 0,Y 141.8,Z 296.661,A -85,B 0,C 180,E1 -27509.853,E2 -27509.853} C_VEL
LIN {X 0,Y 143.673,Z 280.658,A -85,B 0,C 180,E1 -27510.514,E2 -27510.514} C_VEL
LIN {X 0,Y 144.521,Z 270.08,A -85,B 0,C 180,E1 -27510.967,E2 -27510.967} C_VEL
LIN {X 0,Y 142.439,Z 263.614,A -85,B 0,C 180,E1 -27513.197,E2 -27513.197} C_VEL
LIN {X 0,Y 141.37,Z 261.129,A -85,B 0,C 180,E1 -27514.343,E2 -27514.343} C_VEL
LIN {X 0,Y 139.453,Z 258.466,A -85,B 0,C 180,E1 -27516.351,E2 -27516.351} C_VEL
LIN {X 0,Y 137.439,Z 256.752,A -85,B 0,C 180,E1 -27518.567,E2 -27518.567} C_VEL
LIN {X 0,Y 132.77,Z 253.272,A -85,B 0,C 180,E1 -27525.107,E2 -27525.107} C_VEL
LIN {X 0,Y 130.849,Z 249.645,A -85,B 0,C 180,E1 -27529.654,E2 -27529.654} C_VEL
LIN {X 0,Y 129.218,Z 245.465,A -85,B 0,C 180,E1 -27538.442,E2 -27538.442} C_VEL
LIN {X 0,Y 129.211,Z 245.046,A -85,B 0,C 180,E1 -27540,E2 -27540} C_VEL
LIN {X 0,Y 129.225,Z 245.599,A -85,B 0,C 180,E1 -27542.24,E2 -27542.24} C_VEL
LIN {X 0,Y 130.643,Z 249.415,A -85,B 0,C 180,E1 -27550.146,E2 -27550.146} C_VEL
LIN {X 0,Y 131.249,Z 250.477,A -85,B 0,C 180,E1 -27551.837,E2 -27551.837} C_VEL
LIN {X 0,Y 133.357,Z 254.464,A -85,B 0,C 180,E1 -27556.396,E2 -27556.396} C_VEL
LIN {X 0,Y 135.377,Z 258.303,A -85,B 0,C 180,E1 -27559.721,E2 -27559.721} C_VEL
LIN {X 0,Y 138.054,Z 263.698,A -85,B 0,C 180,E1 -27563.352,E2 -27563.352} C_VEL
LIN {X 0,Y 141.208,Z 270.844,A -85,B 0,C 180,E1 -27566.981,E2 -27566.981} C_VEL
LIN {X 0,Y 138.999,Z 291.223,A -85,B 0,C 180,E1 -27567.746,E2 -27567.746} C_VEL
LIN {X 0,Y 136.233,Z 304.644,A -85,B 0,C 180,E1 -27568.539,E2 -27568.539} C_VEL
LIN {X 0,Y 132.57,Z 317.061,A -85,B 0,C 180,E1 -27569.762,E2 -27569.762} C_VEL
LIN {X 0,Y 127.676,Z 329.426,A -85,B 0,C 180,E1 -27571.438,E2 -27571.438} C_VEL
LIN {X 0,Y 122.177,Z 340.45,A -85,B 0,C 180,E1 -27573.479,E2 -27573.479} C_VEL
LIN {X 0,Y 116.866,Z 349.38,A -85,B 0,C 180,E1 -27575.723,E2 -27575.723} C_VEL
LIN {X 0,Y 110.487,Z 358.542,A -85,B 0,C 180,E1 -27578.811,E2 -27578.811} C_VEL
LIN {X 0,Y 103.432,Z 367.473,A -85,B 0,C 180,E1 -27583.11,E2 -27583.11} C_VEL
LIN {X 0,Y 96.913,Z 374.607,A -85,B 0,C 180,E1 -27587.871,E2 -27587.871} C_VEL
LIN {X 0,Y 91.89,Z 379.439,A -85,B 0,C 180,E1 -27592.276,E2 -27592.276} C_VEL
LIN {X 0,Y 86.691,Z 384.132,A -85,B 0,C 180,E1 -27598.2,E2 -27598.2} C_VEL
LIN {X 0,Y 82.548,Z 387.719,A -85,B 0,C 180,E1 -27604.805,E2 -27604.805} C_VEL
LIN {X 0,Y 80.399,Z 389.568,A -85,B 0,C 180,E1 -27609.533,E2 -27609.533} C_VEL
LIN {X 0,Y 78.757,Z 390.956,A -85,B 0,C 180,E1 -27614.472,E2 -27614.472} C_VEL
LIN {X 0,Y 76.996,Z 392.547,A -85,B 0,C 180,E1 -27624.763,E2 -27624.763} C_VEL
LIN {X 0,Y 76.843,Z 392.771,A -85,B 0,C 180,E1 -27630,E2 -27630} C_VEL
LIN {X 0,Y 76.995,Z 392.574,A -85,B 0,C 180,E1 -27635.237,E2 -27635.237} C_VEL
LIN {X 0,Y 77.615,Z 391.988,A -85,B 0,C 180,E1 -27640.434,E2 -27640.434} C_VEL
LIN {X 0,Y 80.353,Z 389.659,A -85,B 0,C 180,E1 -27650.478,E2 -27650.478} C_VEL
LIN {X 0,Y 83.79,Z 386.784,A -85,B 0,C 180,E1 -27657.472,E2 -27657.472} C_VEL
LIN {X 0,Y 88.229,Z 382.886,A -85,B 0,C 180,E1 -27663.889,E2 -27663.889} C_VEL
LIN {X 0,Y 93.776,Z 377.85,A -85,B 0,C 180,E1 -27669.57,E2 -27669.57} C_VEL
LIN {X 0,Y 99.999,Z 371.508,A -85,B 0,C 180,E1 -27674.652,E2 -27674.652} C_VEL
LIN {X 0,Y 106.776,Z 363.58,A -85,B 0,C 180,E1 -27679.194,E2 -27679.194} C_VEL
LIN {X 0,Y 114.219,Z 353.712,A -85,B 0,C 180,E1 -27683.12,E2 -27683.12} C_VEL
LIN {X 0,Y 120.763,Z 343.344,A -85,B 0,C 180,E1 -27686.026,E2 -27686.026} C_VEL
LIN {X 0,Y 126.933,Z 331.649,A -85,B 0,C 180,E1 -27688.35,E2 -27688.35} C_VEL
LIN {X 0,Y 131.83,Z 319.964,A -85,B 0,C 180,E1 -27690.031,E2 -27690.031} C_VEL
LIN {X 0,Y 135.641,Z 307.808,A -85,B 0,C 180,E1 -27691.352,E2 -27691.352} C_VEL
LIN {X 0,Y 138.74,Z 294.313,A -85,B 0,C 180,E1 -27692.275,E2 -27692.275} C_VEL
LIN {X 0,Y 140.648,Z 279.868,A -85,B 0,C 180,E1 -27692.833,E2 -27692.833} C_VEL
LIN {X 0,Y 141.46,Z 271.066,A -85,B 0,C 180,E1 -27693.153,E2 -27693.153} C_VEL
LIN {X 0,Y 138.247,Z 263.738,A -85,B 0,C 180,E1 -27696.871,E2 -27696.871} C_VEL
LIN {X 0,Y 135.41,Z 258.036,A -85,B 0,C 180,E1 -27700.776,E2 -27700.776} C_VEL
LIN {X 0,Y 132.761,Z 253.074,A -85,B 0,C 180,E1 -27705.436,E2 -27705.436} C_VEL
LIN {X 0,Y 131.094,Z 249.729,A -85,B 0,C 180,E1 -27709.576,E2 -27709.576} C_VEL
LIN {X 0,Y 129.536,Z 245.253,A -85,B 0,C 180,E1 -27720,E2 -27720} C_VEL
LIN {X 0,Y 131.247,Z 250.062,A -85,B 0,C 180,E1 -27730.607,E2 -27730.607} C_VEL
LIN {X 0,Y 133.41,Z 254.321,A -85,B 0,C 180,E1 -27735.578,E2 -27735.578} C_VEL
LIN {X 0,Y 135.483,Z 258.214,A -85,B 0,C 180,E1 -27739.065,E2 -27739.065} C_VEL
LIN {X 0,Y 137.934,Z 263.159,A -85,B 0,C 180,E1 -27742.466,E2 -27742.466} C_VEL
LIN {X 0,Y 139.478,Z 267.326,A -85,B 0,C 180,E1 -27744.455,E2 -27744.455} C_VEL
LIN {X 0,Y 141.223,Z 273.129,A -85,B 0,C 180,E1 -27746.608,E2 -27746.608} C_VEL
LIN {X 0,Y 139.173,Z 292.732,A -85,B 0,C 180,E1 -27747.324,E2 -27747.324} C_VEL
LIN {X 0,Y 136.478,Z 306.559,A -85,B 0,C 180,E1 -27748.149,E2 -27748.149} C_VEL
LIN {X 0,Y 132.797,Z 318.852,A -85,B 0,C 180,E1 -27749.165,E2 -27749.165} C_VEL
LIN {X 0,Y 127.792,Z 331.489,A -85,B 0,C 180,E1 -27750.762,E2 -27750.762} C_VEL
LIN {X 0,Y 122.19,Z 342.737,A -85,B 0,C 180,E1 -27752.735,E2 -27752.735} C_VEL
LIN {X 0,Y 116.082,Z 352.865,A -85,B 0,C 180,E1 -27755.181,E2 -27755.181} C_VEL
LIN {X 0,Y 109.555,Z 361.996,A -85,B 0,C 180,E1 -27758.202,E2 -27758.202} C_VEL
LIN {X 0,Y 102.285,Z 370.902,A -85,B 0,C 180,E1 -27762.385,E2 -27762.385} C_VEL
LIN {X 0,Y 96.009,Z 377.822,A -85,B 0,C 180,E1 -27767.056,E2 -27767.056} C_VEL
LIN {X 0,Y 90.87,Z 382.912,A -85,B 0,C 180,E1 -27771.777,E2 -27771.777} C_VEL
LIN {X 0,Y 85.706,Z 387.615,A -85,B 0,C 180,E1 -27777.791,E2 -27777.791} C_VEL
LIN {X 0,Y 81.556,Z 391.21,A -85,B 0,C 180,E1 -27784.478,E2 -27784.478} C_VEL
LIN {X 0,Y 79.567,Z 393.066,A -85,B 0,C 180,E1 -27789.31,E2 -27789.31} C_VEL
LIN {X 0,Y 77.117,Z 395.457,A -85,B 0,C 180,E1 -27799.498,E2 -27799.498} C_VEL
LIN {X 0,Y 76.672,Z 396.066,A -85,B 0,C 180,E1 -27804.741,E2 -27804.741} C_VEL
LIN {X 0,Y 76.731,Z 396.279,A -85,B 0,C 180,E1 -27810,E2 -27810} C_VEL
LIN {X 0,Y 76.707,Z 396.047,A -85,B 0,C 180,E1 -27815.257,E2 -27815.257} C_VEL
LIN {X 0,Y 78.067,Z 394.416,A -85,B 0,C 180,E1 -27825.669,E2 -27825.669} C_VEL
LIN {X 0,Y 79.567,Z 393.003,A -85,B 0,C 180,E1 -27830.69,E2 -27830.69} C_VEL
LIN {X 0,Y 82.821,Z 390.049,A -85,B 0,C 180,E1 -27837.821,E2 -27837.821} C_VEL
LIN {X 0,Y 87.3,Z 386.062,A -85,B 0,C 180,E1 -27844.3,E2 -27844.3} C_VEL
LIN {X 0,Y 93.752,Z 379.933,A -85,B 0,C 180,E1 -27850.99,E2 -27850.99} C_VEL
LIN {X 0,Y 99.987,Z 373.241,A -85,B 0,C 180,E1 -27856.093,E2 -27856.093} C_VEL
LIN {X 0,Y 107.081,Z 364.949,A -85,B 0,C 180,E1 -27860.46,E2 -27860.46} C_VEL
LIN {X 0,Y 113.419,Z 356.44,A -85,B 0,C 180,E1 -27863.662,E2 -27863.662} C_VEL
LIN {X 0,Y 120.086,Z 345.929,A -85,B 0,C 180,E1 -27866.509,E2 -27866.509} C_VEL
LIN {X 0,Y 126.329,Z 334.093,A -85,B 0,C 180,E1 -27868.798,E2 -27868.798} C_VEL
LIN {X 0,Y 131.362,Z 322.152,A -85,B 0,C 180,E1 -27870.388,E2 -27870.388} C_VEL
LIN {X 0,Y 135.384,Z 309.714,A -85,B 0,C 180,E1 -27871.552,E2 -27871.552} C_VEL
LIN {X 0,Y 138.288,Z 296.97,A -85,B 0,C 180,E1 -27872.372,E2 -27872.372} C_VEL
LIN {X 0,Y 140.182,Z 281.88,A -85,B 0,C 180,E1 -27872.989,E2 -27872.989} C_VEL
LIN {X 0,Y 140.973,Z 272.954,A -85,B 0,C 180,E1 -27873.341,E2 -27873.341} C_VEL
LIN {X 0,Y 138.533,Z 264.976,A -85,B 0,C 180,E1 -27876.394,E2 -27876.394} C_VEL
LIN {X 0,Y 136.801,Z 261.135,A -85,B 0,C 180,E1 -27878.629,E2 -27878.629} C_VEL
LIN {X 0,Y 134.217,Z 256.051,A -85,B 0,C 180,E1 -27882.477,E2 -27882.477} C_VEL
LIN {X 0,Y 132.77,Z 253.272,A -85,B 0,C 180,E1 -27885.107,E2 -27885.107} C_VEL
LIN {X 0,Y 131.499,Z 252.257,A -85,B 0,C 180,E1 -27887.568,E2 -27887.568} C_VEL
LIN {X 0,Y 129.658,Z 252.557,A -85,B 0,C 180,E1 -27891.845,E2 -27891.845} C_VEL
LIN {X 0,Y 128.676,Z 253.1,A -85,B 0,C 180,E1 -27895.362,E2 -27895.362} C_VEL
LIN {X 0,Y 128.35,Z 252.804,A -85,B 0,C 180,E1 -27898.012,E2 -27898.012} C_VEL
LIN {X 0,Y 128.333,Z 252.457,A -85,B 0,C 180,E1 -27898.886,E2 -27898.886} C_VEL
LIN {X 0,Y 128.344,Z 252.156,A -85,B 0,C 180,E1 -27900.785,E2 -27900.785} C_VEL
LIN {X 0,Y 129.943,Z 256.994,A -85,B 0,C 180,E1 -27910.742,E2 -27910.742} C_VEL
LIN {X 0,Y 131.847,Z 261.013,A -85,B 0,C 180,E1 -27915.359,E2 -27915.359} C_VEL
LIN {X 0,Y 133.783,Z 264.935,A -85,B 0,C 180,E1 -27918.82,E2 -27918.82} C_VEL
LIN {X 0,Y 136.486,Z 270.921,A -85,B 0,C 180,E1 -27922.753,E2 -27922.753} C_VEL
LIN {X 0,Y 137.843,Z 274.287,A -85,B 0,C 180,E1 -27924.494,E2 -27924.494} C_VEL
LIN {X 0,Y 135.67,Z 292.447,A -85,B 0,C 180,E1 -27925.144,E2 -27925.144} C_VEL
LIN {X 0,Y 132.819,Z 305.469,A -85,B 0,C 180,E1 -27925.903,E2 -27925.903} C_VEL
LIN {X 0,Y 129.202,Z 317.229,A -85,B 0,C 180,E1 -27927.036,E2 -27927.036} C_VEL
LIN {X 0,Y 124.122,Z 329.593,A -85,B 0,C 180,E1 -27928.641,E2 -27928.641} C_VEL
LIN {X 0,Y 118.416,Z 340.616,A -85,B 0,C 180,E1 -27930.618,E2 -27930.618} C_VEL
LIN {X 0,Y 112.873,Z 349.545,A -85,B 0,C 180,E1 -27932.799,E2 -27932.799} C_VEL
LIN {X 0,Y 106.18,Z 358.707,A -85,B 0,C 180,E1 -27935.824,E2 -27935.824} C_VEL
LIN {X 0,Y 98.985,Z 367.338,A -85,B 0,C 180,E1 -27939.933,E2 -27939.933} C_VEL
LIN {X 0,Y 91.775,Z 374.771,A -85,B 0,C 180,E1 -27944.899,E2 -27944.899} C_VEL
LIN {X 0,Y 86.375,Z 379.603,A -85,B 0,C 180,E1 -27949.388,E2 -27949.388} C_VEL
LIN {X 0,Y 80.726,Z 384.296,A -85,B 0,C 180,E1 -27955.536,E2 -27955.536} C_VEL
LIN {X 0,Y 76.167,Z 387.882,A -85,B 0,C 180,E1 -27962.525,E2 -27962.525} C_VEL
LIN {X 0,Y 73.787,Z 389.731,A -85,B 0,C 180,E1 -27967.605,E2 -27967.605} C_VEL
LIN {X 0,Y 71.934,Z 391.119,A -85,B 0,C 180,E1 -27972.956,E2 -27972.956} C_VEL
LIN {X 0,Y 69.929,Z 392.709,A -85,B 0,C 180,E1 -27984.232,E2 -27984.232} C_VEL
LIN {X 0,Y 69.75,Z 392.933,A -85,B 0,C 180,E1 -27990,E2 -27990} C_VEL
LIN {X 0,Y 69.929,Z 392.736,A -85,B 0,C 180,E1 -27995.768,E2 -27995.768} C_VEL
LIN {X 0,Y 70.635,Z 392.15,A -85,B 0,C 180,E1 -28001.478,E2 -28001.478} C_VEL
LIN {X 0,Y 73.749,Z 389.821,A -85,B 0,C 180,E1 -28012.407,E2 -28012.407} C_VEL
LIN {X 0,Y 77.553,Z 386.946,A -85,B 0,C 180,E1 -28019.895,E2 -28019.895} C_VEL
LIN {X 0,Y 82.426,Z 383.047,A -85,B 0,C 180,E1 -28026.644,E2 -28026.644} C_VEL
LIN {X 0,Y 88.418,Z 378.01,A -85,B 0,C 180,E1 -28032.503,E2 -28032.503} C_VEL
LIN {X 0,Y 95.074,Z 371.669,A -85,B 0,C 180,E1 -28037.664,E2 -28037.664} C_VEL
LIN {X 0,Y 102.275,Z 363.74,A -85,B 0,C 180,E1 -28042.208,E2 -28042.208} C_VEL
LIN {X 0,Y 110.113,Z 353.871,A -85,B 0,C 180,E1 -28046.07,E2 -28046.07} C_VEL
LIN {X 0,Y 116.953,Z 343.502,A -85,B 0,C 180,E1 -28048.905,E2 -28048.905} C_VEL
LIN {X 0,Y 123.367,Z 331.807,A -85,B 0,C 180,E1 -28051.15,E2 -28051.15} C_VEL
LIN {X 0,Y 128.438,Z 320.12,A -85,B 0,C 180,E1 -28052.77,E2 -28052.77} C_VEL
LIN {X 0,Y 132.39,Z 307.961,A -85,B 0,C 180,E1 -28054.044,E2 -28054.044} C_VEL
LIN {X 0,Y 135.475,Z 295.041,A -85,B 0,C 180,E1 -28054.892,E2 -28054.892} C_VEL
LIN {X 0,Y 137.322,Z 282.245,A -85,B 0,C 180,E1 -28055.398,E2 -28055.398} C_VEL
LIN {X 0,Y 138.074,Z 274.471,A -85,B 0,C 180,E1 -28055.671,E2 -28055.671} C_VEL
LIN {X 0,Y 135.502,Z 268.269,A -85,B 0,C 180,E1 -28059.109,E2 -28059.109} C_VEL
LIN {X 0,Y 133.006,Z 262.994,A -85,B 0,C 180,E1 -28063.105,E2 -28063.105} C_VEL
LIN {X 0,Y 131.343,Z 259.66,A -85,B 0,C 180,E1 -28066.461,E2 -28066.461} C_VEL
LIN {X 0,Y 129.833,Z 256.459,A -85,B 0,C 180,E1 -28070.654,E2 -28070.654} C_VEL
LIN {X 0,Y 128.647,Z 252.493,A -85,B 0,C 180,E1 -28080,E2 -28080} C_VEL
LIN {X 0,Y 130.095,Z 256.97,A -85,B 0,C 180,E1 -28089.915,E2 -28089.915} C_VEL
LIN {X 0,Y 131.982,Z 260.943,A -85,B 0,C 180,E1 -28094.651,E2 -28094.651} C_VEL
LIN {X 0,Y 134.126,Z 265.295,A -85,B 0,C 180,E1 -28098.522,E2 -28098.522} C_VEL
LIN {X 0,Y 136.276,Z 270.253,A -85,B 0,C 180,E1 -28101.734,E2 -28101.734} C_VEL
LIN {X 0,Y 137.895,Z 275.87,A -85,B 0,C 180,E1 -28104.062,E2 -28104.062} C_VEL
LIN {X 0,Y 135.845,Z 293.861,A -85,B 0,C 180,E1 -28104.718,E2 -28104.718} C_VEL
LIN {X 0,Y 133.112,Z 307.062,A -85,B 0,C 180,E1 -28105.499,E2 -28105.499} C_VEL
LIN {X 0,Y 129.493,Z 318.697,A -85,B 0,C 180,E1 -28106.427,E2 -28106.427} C_VEL
LIN {X 0,Y 124.317,Z 331.332,A -85,B 0,C 180,E1 -28107.954,E2 -28107.954} C_VEL
LIN {X 0,Y 118.491,Z 342.578,A -85,B 0,C 180,E1 -28109.838,E2 -28109.838} C_VEL
LIN {X 0,Y 112.129,Z 352.706,A -85,B 0,C 180,E1 -28112.206,E2 -28112.206} C_VEL
LIN {X 0,Y 105.314,Z 361.837,A -85,B 0,C 180,E1 -28115.166,E2 -28115.166} C_VEL
LIN {X 0,Y 97.63,Z 370.742,A -85,B 0,C 180,E1 -28119.299,E2 -28119.299} C_VEL
LIN {X 0,Y 90.314,Z 378.229,A -85,B 0,C 180,E1 -28124.455,E2 -28124.455} C_VEL
LIN {X 0,Y 85.399,Z 382.751,A -85,B 0,C 180,E1 -28128.825,E2 -28128.825} C_VEL
LIN {X 0,Y 79.769,Z 387.454,A -85,B 0,C 180,E1 -28135.063,E2 -28135.063} C_VEL
LIN {X 0,Y 75.181,Z 391.047,A -85,B 0,C 180,E1 -28142.134,E2 -28142.134} C_VEL
LIN {X 0,Y 72.935,Z 392.904,A -85,B 0,C 180,E1 -28147.329,E2 -28147.329} C_VEL
LIN {X 0,Y 70.139,Z 395.294,A -85,B 0,C 180,E1 -28158.44,E2 -28158.44} C_VEL
LIN {X 0,Y 69.591,Z 395.903,A -85,B 0,C 180,E1 -28164.204,E2 -28164.204} C_VEL
LIN {X 0,Y 69.641,Z 396.117,A -85,B 0,C 180,E1 -28170,E2 -28170} C_VEL
LIN {X 0,Y 69.62,Z 395.884,A -85,B 0,C 180,E1 -28175.794,E2 -28175.794} C_VEL
LIN {X 0,Y 70.144,Z 395.263,A -85,B 0,C 180,E1 -28181.56,E2 -28181.56} C_VEL
LIN {X 0,Y 71.233,Z 394.253,A -85,B 0,C 180,E1 -28187.217,E2 -28187.217} C_VEL
LIN {X 0,Y 72.935,Z 392.84,A -85,B 0,C 180,E1 -28192.671,E2 -28192.671} C_VEL
LIN {X 0,Y 76.593,Z 389.886,A -85,B 0,C 180,E1 -28200.309,E2 -28200.309} C_VEL
LIN {X 0,Y 81.499,Z 385.897,A -85,B 0,C 180,E1 -28207.131,E2 -28207.131} C_VEL
LIN {X 0,Y 87.456,Z 380.772,A -85,B 0,C 180,E1 -28213.084,E2 -28213.084} C_VEL
LIN {X 0,Y 93.988,Z 374.312,A -85,B 0,C 180,E1 -28218.396,E2 -28218.396} C_VEL
LIN {X 0,Y 101.396,Z 366.273,A -85,B 0,C 180,E1 -28222.853,E2 -28222.853} C_VEL
LIN {X 0,Y 107.986,Z 358.08,A -85,B 0,C 180,E1 -28226.078,E2 -28226.078} C_VEL
LIN {X 0,Y 114.889,Z 348.088,A -85,B 0,C 180,E1 -28228.916,E2 -28228.916} C_VEL
LIN {X 0,Y 121.354,Z 336.787,A -85,B 0,C 180,E1 -28231.156,E2 -28231.156} C_VEL
LIN {X 0,Y 126.514,Z 325.711,A -85,B 0,C 180,E1 -28232.725,E2 -28232.725} C_VEL
LIN {X 0,Y 130.999,Z 313.407,A -85,B 0,C 180,E1 -28233.978,E2 -28233.978} C_VEL
LIN {X 0,Y 134.485,Z 300.041,A -85,B 0,C 180,E1 -28234.864,E2 -28234.864} C_VEL
LIN {X 0,Y 136.637,Z 286.445,A -85,B 0,C 180,E1 -28235.461,E2 -28235.461} C_VEL
LIN {X 0,Y 137.64,Z 275.647,A -85,B 0,C 180,E1 -28235.89,E2 -28235.89} C_VEL
LIN {X 0,Y 135.719,Z 269.19,A -85,B 0,C 180,E1 -28238.648,E2 -28238.648} C_VEL
LIN {X 0,Y 132.975,Z 263.153,A -85,B 0,C 180,E1 -28242.923,E2 -28242.923} C_VEL
LIN {X 0,Y 131.003,Z 259.317,A -85,B 0,C 180,E1 -28246.823,E2 -28246.823} C_VEL
LIN {X 0,Y 129.615,Z 256.365,A -85,B 0,C 180,E1 -28250.638,E2 -28250.638} C_VEL
LIN {X 0,Y 128.333,Z 252.457,A -85,B 0,C 180,E1 -28258.886,E2 -28258.886} C_VEL
LIN {X 0,Y 128.28,Z 252.626,A -85,B 0,C 180,E1 -28260.296,E2 -28260.296} C_VEL
LIN {X 0,Y 128.097,Z 254.708,A -85,B 0,C 180,E1 -28262.128,E2 -28262.128} C_VEL
LIN {X 0,Y 127.831,Z 260.863,A -85,B 0,C 180,E1 -28265.564,E2 -28265.564} C_VEL
LIN {X 0,Y 128.046,Z 262.52,A -85,B 0,C 180,E1 -28267.283,E2 -28267.283} C_VEL
LIN {X 0,Y 128.749,Z 263.721,A -85,B 0,C 180,E1 -28269.861,E2 -28269.861} C_VEL
LIN {X 0,Y 130.36,Z 267.469,A -85,B 0,C 180,E1 -28274.24,E2 -28274.24} C_VEL
LIN {X 0,Y 132.013,Z 271.141,A -85,B 0,C 180,E1 -28277.535,E2 -28277.535} C_VEL
LIN {X 0,Y 134.304,Z 276.675,A -85,B 0,C 180,E1 -28281.251,E2 -28281.251} C_VEL
LIN {X 0,Y 134.698,Z 277.764,A -85,B 0,C 180,E1 -28281.837,E2 -28281.837} C_VEL
LIN {X 0,Y 132.632,Z 293.652,A -85,B 0,C 180,E1 -28282.409,E2 -28282.409} C_VEL
LIN {X 0,Y 129.875,Z 305.64,A -85,B 0,C 180,E1 -28283.085,E2 -28283.085} C_VEL
LIN {X 0,Y 126.069,Z 317.576,A -85,B 0,C 180,E1 -28284.184,E2 -28284.184} C_VEL
LIN {X 0,Y 120.886,Z 329.76,A -85,B 0,C 180,E1 -28285.693,E2 -28285.693} C_VEL
LIN {X 0,Y 114.962,Z 340.782,A -85,B 0,C 180,E1 -28287.572,E2 -28287.572} C_VEL
LIN {X 0,Y 109.187,Z 349.711,A -85,B 0,C 180,E1 -28289.664,E2 -28289.664} C_VEL
LIN {X 0,Y 102.181,Z 358.872,A -85,B 0,C 180,E1 -28292.59,E2 -28292.59} C_VEL
LIN {X 0,Y 94.15,Z 367.959,A -85,B 0,C 180,E1 -28296.885,E2 -28296.885} C_VEL
LIN {X 0,Y 86.908,Z 374.935,A -85,B 0,C 180,E1 -28301.581,E2 -28301.581} C_VEL
LIN {X 0,Y 81.113,Z 379.767,A -85,B 0,C 180,E1 -28306.12,E2 -28306.12} C_VEL
LIN {X 0,Y 74.97,Z 384.46,A -85,B 0,C 180,E1 -28312.458,E2 -28312.458} C_VEL
LIN {X 0,Y 69.937,Z 388.045,A -85,B 0,C 180,E1 -28319.838,E2 -28319.838} C_VEL
LIN {X 0,Y 67.281,Z 389.894,A -85,B 0,C 180,E1 -28325.302,E2 -28325.302} C_VEL
LIN {X 0,Y 65.182,Z 391.281,A -85,B 0,C 180,E1 -28331.127,E2 -28331.127} C_VEL
LIN {X 0,Y 62.887,Z 392.871,A -85,B 0,C 180,E1 -28343.583,E2 -28343.583} C_VEL
LIN {X 0,Y 62.677,Z 393.094,A -85,B 0,C 180,E1 -28350,E2 -28350} C_VEL
LIN {X 0,Y 62.887,Z 392.898,A -85,B 0,C 180,E1 -28356.416,E2 -28356.416} C_VEL
LIN {X 0,Y 63.698,Z 392.311,A -85,B 0,C 180,E1 -28362.748,E2 -28362.748} C_VEL
LIN {X 0,Y 67.221,Z 389.983,A -85,B 0,C 180,E1 -28374.721,E2 -28374.721} C_VEL
LIN {X 0,Y 71.482,Z 387.107,A -85,B 0,C 180,E1 -28382.734,E2 -28382.734} C_VEL
LIN {X 0,Y 76.846,Z 383.208,A -85,B 0,C 180,E1 -28389.805,E2 -28389.805} C_VEL
LIN {X 0,Y 83.323,Z 378.171,A -85,B 0,C 180,E1 -28395.802,E2 -28395.802} C_VEL
LIN {X 0,Y 90.443,Z 371.829,A -85,B 0,C 180,E1 -28400.992,E2 -28400.992} C_VEL
LIN {X 0,Y 98.075,Z 363.9,A -85,B 0,C 180,E1 -28405.495,E2 -28405.495} C_VEL
LIN {X 0,Y 106.311,Z 354.031,A -85,B 0,C 180,E1 -28409.249,E2 -28409.249} C_VEL
LIN {X 0,Y 113.461,Z 343.66,A -85,B 0,C 180,E1 -28411.966,E2 -28411.966} C_VEL
LIN {X 0,Y 120.112,Z 331.964,A -85,B 0,C 180,E1 -28414.108,E2 -28414.108} C_VEL
LIN {X 0,Y 125.351,Z 320.275,A -85,B 0,C 180,E1 -28415.654,E2 -28415.654} C_VEL
LIN {X 0,Y 129.567,Z 307.714,A -85,B 0,C 180,E1 -28416.892,E2 -28416.892} C_VEL
LIN {X 0,Y 132.629,Z 295.191,A -85,B 0,C 180,E1 -28417.66,E2 -28417.66} C_VEL
LIN {X 0,Y 134.528,Z 282.384,A -85,B 0,C 180,E1 -28418.142,E2 -28418.142} C_VEL
LIN {X 0,Y 134.923,Z 277.863,A -85,B 0,C 180,E1 -28418.359,E2 -28418.359} C_VEL
LIN {X 0,Y 132.653,Z 272.152,A -85,B 0,C 180,E1 -28421.964,E2 -28421.964} C_VEL
LIN {X 0,Y 130.941,Z 268.4,A -85,B 0,C 180,E1 -28425.229,E2 -28425.229} C_VEL
LIN {X 0,Y 129.894,Z 266.081,A -85,B 0,C 180,E1 -28427.699,E2 -28427.699} C_VEL
LIN {X 0,Y 128.788,Z 263.39,A -85,B 0,C 180,E1 -28431.171,E2 -28431.171} C_VEL
LIN {X 0,Y 127.762,Z 259.707,A -85,B 0,C 180,E1 -28440,E2 -28440} C_VEL
LIN {X 0,Y 128.966,Z 263.848,A -85,B 0,C 180,E1 -28449.211,E2 -28449.211} C_VEL
LIN {X 0,Y 130.511,Z 267.407,A -85,B 0,C 180,E1 -28453.527,E2 -28453.527} C_VEL
LIN {X 0,Y 132.369,Z 271.534,A -85,B 0,C 180,E1 -28457.266,E2 -28457.266} C_VEL
LIN {X 0,Y 134.089,Z 275.91,A -85,B 0,C 180,E1 -28460.148,E2 -28460.148} C_VEL
LIN {X 0,Y 134.833,Z 278.784,A -85,B 0,C 180,E1 -28461.399,E2 -28461.399} C_VEL
LIN {X 0,Y 132.978,Z 294.078,A -85,B 0,C 180,E1 -28461.962,E2 -28461.962} C_VEL
LIN {X 0,Y 130.219,Z 306.909,A -85,B 0,C 180,E1 -28462.683,E2 -28462.683} C_VEL
LIN {X 0,Y 126.492,Z 318.541,A -85,B 0,C 180,E1 -28463.545,E2 -28463.545} C_VEL
LIN {X 0,Y 121.154,Z 331.175,A -85,B 0,C 180,E1 -28464.99,E2 -28464.99} C_VEL
LIN {X 0,Y 115.126,Z 342.42,A -85,B 0,C 180,E1 -28466.774,E2 -28466.774} C_VEL
LIN {X 0,Y 108.509,Z 352.546,A -85,B 0,C 180,E1 -28469.029,E2 -28469.029} C_VEL
LIN {X 0,Y 101.39,Z 361.677,A -85,B 0,C 180,E1 -28471.884,E2 -28471.884} C_VEL
LIN {X 0,Y 93.279,Z 370.581,A -85,B 0,C 180,E1 -28475.91,E2 -28475.91} C_VEL
LIN {X 0,Y 87.016,Z 376.637,A -85,B 0,C 180,E1 -28479.893,E2 -28479.893} C_VEL
LIN {X 0,Y 80.184,Z 382.59,A -85,B 0,C 180,E1 -28485.478,E2 -28485.478} C_VEL
LIN {X 0,Y 74.042,Z 387.292,A -85,B 0,C 180,E1 -28491.905,E2 -28491.905} C_VEL
LIN {X 0,Y 68.961,Z 390.885,A -85,B 0,C 180,E1 -28499.366,E2 -28499.366} C_VEL
LIN {X 0,Y 66.396,Z 392.741,A -85,B 0,C 180,E1 -28504.951,E2 -28504.951} C_VEL
LIN {X 0,Y 64.464,Z 394.135,A -85,B 0,C 180,E1 -28510.91,E2 -28510.91} C_VEL
LIN {X 0,Y 63.176,Z 395.132,A -85,B 0,C 180,E1 -28517.145,E2 -28517.145} C_VEL
LIN {X 0,Y 62.532,Z 395.741,A -85,B 0,C 180,E1 -28523.547,E2 -28523.547} C_VEL
LIN {X 0,Y 62.54,Z 395.955,A -85,B 0,C 180,E1 -28530,E2 -28530} C_VEL
LIN {X 0,Y 62.555,Z 395.722,A -85,B 0,C 180,E1 -28536.451,E2 -28536.451} C_VEL
LIN {X 0,Y 64.469,Z 394.09,A -85,B 0,C 180,E1 -28549.089,E2 -28549.089} C_VEL
LIN {X 0,Y 66.396,Z 392.676,A -85,B 0,C 180,E1 -28555.05,E2 -28555.05} C_VEL
LIN {X 0,Y 70.538,Z 389.722,A -85,B 0,C 180,E1 -28563.229,E2 -28563.229} C_VEL
LIN {X 0,Y 75.932,Z 385.733,A -85,B 0,C 180,E1 -28570.383,E2 -28570.383} C_VEL
LIN {X 0,Y 81.733,Z 381.148,A -85,B 0,C 180,E1 -28575.912,E2 -28575.912} C_VEL
LIN {X 0,Y 89.416,Z 374.147,A -85,B 0,C 180,E1 -28581.813,E2 -28581.813} C_VEL
LIN {X 0,Y 97.27,Z 366.108,A -85,B 0,C 180,E1 -28586.192,E2 -28586.192} C_VEL
LIN {X 0,Y 104.19,Z 357.915,A -85,B 0,C 180,E1 -28589.321,E2 -28589.321} C_VEL
LIN {X 0,Y 111.387,Z 347.923,A -85,B 0,C 180,E1 -28592.047,E2 -28592.047} C_VEL
LIN {X 0,Y 118.096,Z 336.62,A -85,B 0,C 180,E1 -28594.171,E2 -28594.171} C_VEL
LIN {X 0,Y 123.418,Z 325.543,A -85,B 0,C 180,E1 -28595.66,E2 -28595.66} C_VEL
LIN {X 0,Y 128.05,Z 313.238,A -85,B 0,C 180,E1 -28596.826,E2 -28596.826} C_VEL
LIN {X 0,Y 131.513,Z 300.377,A -85,B 0,C 180,E1 -28597.643,E2 -28597.643} C_VEL
LIN {X 0,Y 133.76,Z 286.921,A -85,B 0,C 180,E1 -28598.207,E2 -28598.207} C_VEL
LIN {X 0,Y 134.569,Z 278.548,A -85,B 0,C 180,E1 -28598.557,E2 -28598.557} C_VEL
LIN {X 0,Y 133.383,Z 274.364,A -85,B 0,C 180,E1 -28600.527,E2 -28600.527} C_VEL
LIN {X 0,Y 131.06,Z 268.981,A -85,B 0,C 180,E1 -28604.647,E2 -28604.647} C_VEL
LIN {X 0,Y 129.634,Z 265.865,A -85,B 0,C 180,E1 -28607.873,E2 -28607.873} C_VEL
LIN {X 0,Y 128.505,Z 263.196,A -85,B 0,C 180,E1 -28611.35,E2 -28611.35} C_VEL
LIN {X 0,Y 127.476,Z 259.176,A -85,B 0,C 180,E1 -28620,E2 -28620} C_VEL
LIN {X 0,Y 127.448,Z 260.155,A -85,B 0,C 180,E1 -28622.37,E2 -28622.37} C_VEL
LIN {X 0,Y 128.046,Z 262.52,A -85,B 0,C 180,E1 -28627.283,E2 -28627.283} C_VEL
LIN {X 0,Y 128.6,Z 264.546,A -85,B 0,C 180,E1 -28629.74,E2 -28629.74} C_VEL
LIN {X 0,Y 129.141,Z 267.736,A -85,B 0,C 180,E1 -28631.957,E2 -28631.957} C_VEL
LIN {X 0,Y 131.632,Z 280.806,A -85,B 0,C 180,E1 -28638.698,E2 -28638.698} C_VEL
LIN {X 0,Y 131.851,Z 281.39,A -85,B 0,C 180,E1 -28639.076,E2 -28639.076} C_VEL
LIN {X 0,Y 129.964,Z 294.543,A -85,B 0,C 180,E1 -28639.549,E2 -28639.549} C_VEL
LIN {X 0,Y 126.682,Z 307.742,A -85,B 0,C 180,E1 -28640.286,E2 -28640.286} C_VEL
LIN {X 0,Y 122.483,Z 319.92,A -85,B 0,C 180,E1 -28641.396,E2 -28641.396} C_VEL
LIN {X 0,Y 117.224,Z 331.487,A -85,B 0,C 180,E1 -28642.812,E2 -28642.812} C_VEL
LIN {X 0,Y 110.349,Z 343.298,A -85,B 0,C 180,E1 -28644.83,E2 -28644.83} C_VEL
LIN {X 0,Y 102.897,Z 353.774,A -85,B 0,C 180,E1 -28647.387,E2 -28647.387} C_VEL
LIN {X 0,Y 95.707,Z 362.248,A -85,B 0,C 180,E1 -28650.364,E2 -28650.364} C_VEL
LIN {X 0,Y 87.884,Z 370.19,A -85,B 0,C 180,E1 -28654.459,E2 -28654.459} C_VEL
LIN {X 0,Y 81.057,Z 376.125,A -85,B 0,C 180,E1 -28658.708,E2 -28658.708} C_VEL
LIN {X 0,Y 73.834,Z 381.62,A -85,B 0,C 180,E1 -28664.447,E2 -28664.447} C_VEL
LIN {X 0,Y 67.472,Z 385.931,A -85,B 0,C 180,E1 -28671.32,E2 -28671.32} C_VEL
LIN {X 0,Y 63.897,Z 388.208,A -85,B 0,C 180,E1 -28676.636,E2 -28676.636} C_VEL
LIN {X 0,Y 60.885,Z 390.057,A -85,B 0,C 180,E1 -28682.501,E2 -28682.501} C_VEL
LIN {X 0,Y 58.498,Z 391.444,A -85,B 0,C 180,E1 -28688.874,E2 -28688.874} C_VEL
LIN {X 0,Y 55.839,Z 393.033,A -85,B 0,C 180,E1 -28702.769,E2 -28702.769} C_VEL
LIN {X 0,Y 55.593,Z 393.256,A -85,B 0,C 180,E1 -28710,E2 -28710} C_VEL
LIN {X 0,Y 55.838,Z 393.06,A -85,B 0,C 180,E1 -28717.23,E2 -28717.23} C_VEL
LIN {X 0,Y 56.789,Z 392.473,A -85,B 0,C 180,E1 -28724.33,E2 -28724.33} C_VEL
LIN {X 0,Y 60.836,Z 390.145,A -85,B 0,C 180,E1 -28737.522,E2 -28737.522} C_VEL
LIN {X 0,Y 65.619,Z 387.269,A -85,B 0,C 180,E1 -28746.09,E2 -28746.09} C_VEL
LIN {X 0,Y 71.539,Z 383.369,A -85,B 0,C 180,E1 -28753.446,E2 -28753.446} C_VEL
LIN {X 0,Y 78.542,Z 378.332,A -85,B 0,C 180,E1 -28759.516,E2 -28759.516} C_VEL
LIN {X 0,Y 86.15,Z 371.989,A -85,B 0,C 180,E1 -28764.664,E2 -28764.664} C_VEL
LIN {X 0,Y 94.23,Z 364.06,A -85,B 0,C 180,E1 -28769.06,E2 -28769.06} C_VEL
LIN {X 0,Y 102.868,Z 354.19,A -85,B 0,C 180,E1 -28772.643,E2 -28772.643} C_VEL
LIN {X 0,Y 110.304,Z 343.818,A -85,B 0,C 180,E1 -28775.221,E2 -28775.221} C_VEL
LIN {X 0,Y 117.184,Z 332.121,A -85,B 0,C 180,E1 -28777.235,E2 -28777.235} C_VEL
LIN {X 0,Y 122.534,Z 320.602,A -85,B 0,C 180,E1 -28778.655,E2 -28778.655} C_VEL
LIN {X 0,Y 126.955,Z 307.867,A -85,B 0,C 180,E1 -28779.833,E2 -28779.833} C_VEL
LIN {X 0,Y 130.223,Z 294.763,A -85,B 0,C 180,E1 -28780.576,E2 -28780.576} C_VEL
LIN {X 0,Y 132.115,Z 281.588,A -85,B 0,C 180,E1 -28781.073,E2 -28781.073} C_VEL
LIN {X 0,Y 130.075,Z 276.167,A -85,B 0,C 180,E1 -28785.029,E2 -28785.029} C_VEL
LIN {X 0,Y 128.511,Z 272.477,A -85,B 0,C 180,E1 -28788.965,E2 -28788.965} C_VEL
LIN {X 0,Y 127.647,Z 270.189,A -85,B 0,C 180,E1 -28792.088,E2 -28792.088} C_VEL
LIN {X 0,Y 126.881,Z 266.882,A -85,B 0,C 180,E1 -28800,E2 -28800} C_VEL
LIN {X 0,Y 127.876,Z 270.745,A -85,B 0,C 180,E1 -28808.558,E2 -28808.558} C_VEL
LIN {X 0,Y 129.239,Z 274.245,A -85,B 0,C 180,E1 -28812.763,E2 -28812.763} C_VEL
LIN {X 0,Y 130.849,Z 278.13,A -85,B 0,C 180,E1 -28816.302,E2 -28816.302} C_VEL
LIN {X 0,Y 132.061,Z 281.827,A -85,B 0,C 180,E1 -28818.621,E2 -28818.621} C_VEL
LIN {X 0,Y 131.227,Z 289.197,A -85,B 0,C 180,E1 -28818.89,E2 -28818.89} C_VEL
LIN {X 0,Y 128.711,Z 302.683,A -85,B 0,C 180,E1 -28819.512,E2 -28819.512} C_VEL
LIN {X 0,Y 124.965,Z 315.249,A -85,B 0,C 180,E1 -28820.311,E2 -28820.311} C_VEL
LIN {X 0,Y 119.892,Z 327.78,A -85,B 0,C 180,E1 -28821.475,E2 -28821.475} C_VEL
LIN {X 0,Y 113.665,Z 339.676,A -85,B 0,C 180,E1 -28823.113,E2 -28823.113} C_VEL
LIN {X 0,Y 106.745,Z 350.288,A -85,B 0,C 180,E1 -28825.139,E2 -28825.139} C_VEL
LIN {X 0,Y 99.274,Z 359.854,A -85,B 0,C 180,E1 -28827.759,E2 -28827.759} C_VEL
LIN {X 0,Y 90.678,Z 369.063,A -85,B 0,C 180,E1 -28831.51,E2 -28831.51} C_VEL
LIN {X 0,Y 82.618,Z 376.473,A -85,B 0,C 180,E1 -28836.087,E2 -28836.087} C_VEL
LIN {X 0,Y 75.264,Z 382.428,A -85,B 0,C 180,E1 -28841.667,E2 -28841.667} C_VEL
LIN {X 0,Y 68.578,Z 387.13,A -85,B 0,C 180,E1 -28848.231,E2 -28848.231} C_VEL
LIN {X 0,Y 62.94,Z 390.724,A -85,B 0,C 180,E1 -28856.061,E2 -28856.061} C_VEL
LIN {X 0,Y 59.998,Z 392.578,A -85,B 0,C 180,E1 -28862.06,E2 -28862.06} C_VEL
LIN {X 0,Y 57.776,Z 393.972,A -85,B 0,C 180,E1 -28868.597,E2 -28868.597} C_VEL
LIN {X 0,Y 56.266,Z 394.97,A -85,B 0,C 180,E1 -28875.534,E2 -28875.534} C_VEL
LIN {X 0,Y 55.474,Z 395.579,A -85,B 0,C 180,E1 -28882.722,E2 -28882.722} C_VEL
LIN {X 0,Y 55.458,Z 395.793,A -85,B 0,C 180,E1 -28890,E2 -28890} C_VEL
LIN {X 0,Y 55.513,Z 395.56,A -85,B 0,C 180,E1 -28897.274,E2 -28897.274} C_VEL
LIN {X 0,Y 57.78,Z 393.926,A -85,B 0,C 180,E1 -28911.402,E2 -28911.402} C_VEL
LIN {X 0,Y 59.998,Z 392.512,A -85,B 0,C 180,E1 -28917.94,E2 -28917.94} C_VEL
LIN {X 0,Y 64.704,Z 389.559,A -85,B 0,C 180,E1 -28926.684,E2 -28926.684} C_VEL
LIN {X 0,Y 70.654,Z 385.569,A -85,B 0,C 180,E1 -28934.131,E2 -28934.131} C_VEL
LIN {X 0,Y 77.936,Z 380.154,A -85,B 0,C 180,E1 -28940.633,E2 -28940.633} C_VEL
LIN {X 0,Y 86.55,Z 372.747,A -85,B 0,C 180,E1 -28946.338,E2 -28946.338} C_VEL
LIN {X 0,Y 94.908,Z 364.453,A -85,B 0,C 180,E1 -28950.47,E2 -28950.47} C_VEL
LIN {X 0,Y 102.233,Z 355.943,A -85,B 0,C 180,E1 -28953.34,E2 -28953.34} C_VEL
LIN {X 0,Y 109.78,Z 345.431,A -85,B 0,C 180,E1 -28955.821,E2 -28955.821} C_VEL
LIN {X 0,Y 116.725,Z 333.592,A -85,B 0,C 180,E1 -28957.778,E2 -28957.778} C_VEL
LIN {X 0,Y 122.158,Z 321.876,A -85,B 0,C 180,E1 -28959.077,E2 -28959.077} C_VEL
LIN {X 0,Y 126.66,Z 309.106,A -85,B 0,C 180,E1 -28960.064,E2 -28960.064} C_VEL
LIN {X 0,Y 129.741,Z 296.749,A -85,B 0,C 180,E1 -28960.706,E2 -28960.706} C_VEL
LIN {X 0,Y 131.702,Z 283.048,A -85,B 0,C 180,E1 -28961.206,E2 -28961.206} C_VEL
LIN {X 0,Y 131.794,Z 281.529,A -85,B 0,C 180,E1 -28961.34,E2 -28961.34} C_VEL
LIN {X 0,Y 130.694,Z 278.298,A -85,B 0,C 180,E1 -28963.401,E2 -28963.401} C_VEL
LIN {X 0,Y 129.18,Z 274.584,A -85,B 0,C 180,E1 -28966.63,E2 -28966.63} C_VEL
LIN {X 0,Y 128.188,Z 272.194,A -85,B 0,C 180,E1 -28969.287,E2 -28969.287} C_VEL
LIN {X 0,Y 127.362,Z 269.976,A -85,B 0,C 180,E1 -28972.27,E2 -28972.27} C_VEL
LIN {X 0,Y 126.599,Z 266.315,A -85,B 0,C 180,E1 -28980.398,E2 -28980.398} C_VEL
LIN {X 0,Y 127.644,Z 270.671,A -85,B 0,C 180,E1 -28989.208,E2 -28989.208} C_VEL
LIN {X 0,Y 129.046,Z 274.222,A -85,B 0,C 180,E1 -28993.401,E2 -28993.401} C_VEL
LIN {X 0,Y 130.715,Z 278.309,A -85,B 0,C 180,E1 -28996.999,E2 -28996.999} C_VEL
LIN {X 0,Y 131.632,Z 280.806,A -85,B 0,C 180,E1 -28998.698,E2 -28998.698} C_VEL
LIN {X 0,Y 131.908,Z 282.874,A -85,B 0,C 180,E1 -28999.387,E2 -28999.387} C_VEL
LIN {X 0,Y 131.65,Z 286.427,A -85,B 0,C 180,E1 -28999.721,E2 -28999.721} C_VEL
LIN {X 0,Y 130.68,Z 291.016,A -85,B 0,C 180,E1 -28999.518,E2 -28999.518} C_VEL
LIN {X 0,Y 125.708,Z 304.828,A -85,B 0,C 180,E1 -28997.554,E2 -28997.554} C_VEL
LIN {X 0,Y 123.757,Z 310.103,A -85,B 0,C 180,E1 -28997.394,E2 -28997.394} C_VEL
LIN {X 0,Y 123.394,Z 311.16,A -85,B 0,C 180,E1 -28997.462,E2 -28997.462} C_VEL
LIN {X 0,Y 118.616,Z 323.449,A -85,B 0,C 180,E1 -28998.558,E2 -28998.558} C_VEL
LIN {X 0,Y 112.298,Z 335.929,A -85,B 0,C 180,E1 -29000.157,E2 -29000.157} C_VEL
LIN {X 0,Y 106.016,Z 345.783,A -85,B 0,C 180,E1 -29001.862,E2 -29001.862} C_VEL
LIN {X 0,Y 98.309,Z 355.74,A -85,B 0,C 180,E1 -29004.289,E2 -29004.289} C_VEL
LIN {X 0,Y 90.866,Z 363.892,A -85,B 0,C 180,E1 -29007.194,E2 -29007.194} C_VEL
LIN {X 0,Y 82.308,Z 371.879,A -85,B 0,C 180,E1 -29011.365,E2 -29011.365} C_VEL
LIN {X 0,Y 74.166,Z 378.286,A -85,B 0,C 180,E1 -29016.345,E2 -29016.345} C_VEL
LIN {X 0,Y 66.602,Z 383.37,A -85,B 0,C 180,E1 -29022.382,E2 -29022.382} C_VEL
LIN {X 0,Y 60.029,Z 387.312,A -85,B 0,C 180,E1 -29029.915,E2 -29029.915} C_VEL
LIN {X 0,Y 54.677,Z 390.22,A -85,B 0,C 180,E1 -29039.06,E2 -29039.06} C_VEL
LIN {X 0,Y 51.937,Z 391.607,A -85,B 0,C 180,E1 -29046.049,E2 -29046.049} C_VEL
LIN {X 0,Y 48.82,Z 393.195,A -85,B 0,C 180,E1 -29061.723,E2 -29061.723} C_VEL
LIN {X 0,Y 48.497,Z 393.418,A -85,B 0,C 180,E1 -29070,E2 -29070} C_VEL
LIN {X 0,Y 48.819,Z 393.221,A -85,B 0,C 180,E1 -29078.277,E2 -29078.277} C_VEL
LIN {X 0,Y 51.896,Z 391.667,A -85,B 0,C 180,E1 -29093.971,E2 -29093.971} C_VEL
LIN {X 0,Y 54.637,Z 390.306,A -85,B 0,C 180,E1 -29100.965,E2 -29100.965} C_VEL
LIN {X 0,Y 60.006,Z 387.431,A -85,B 0,C 180,E1 -29110.103,E2 -29110.103} C_VEL
LIN {X 0,Y 66.569,Z 383.53,A -85,B 0,C 180,E1 -29117.647,E2 -29117.647} C_VEL
LIN {X 0,Y 74.132,Z 378.492,A -85,B 0,C 180,E1 -29123.69,E2 -29123.69} C_VEL
LIN {X 0,Y 82.245,Z 372.15,A -85,B 0,C 180,E1 -29128.706,E2 -29128.706} C_VEL
LIN {X 0,Y 90.787,Z 364.22,A -85,B 0,C 180,E1 -29132.902,E2 -29132.902} C_VEL
LIN {X 0,Y 98.274,Z 356.129,A -85,B 0,C 180,E1 -29135.756,E2 -29135.756} C_VEL
LIN {X 0,Y 105.957,Z 346.256,A -85,B 0,C 180,E1 -29138.216,E2 -29138.216} C_VEL
LIN {X 0,Y 113.03,Z 335.126,A -85,B 0,C 180,E1 -29140.125,E2 -29140.125} C_VEL
LIN {X 0,Y 119.319,Z 322.646,A -85,B 0,C 180,E1 -29141.616,E2 -29141.616} C_VEL
LIN {X 0,Y 123.821,Z 310.845,A -85,B 0,C 180,E1 -29142.691,E2 -29142.691} C_VEL
LIN {X 0,Y 127.293,Z 298.309,A -85,B 0,C 180,E1 -29143.415,E2 -29143.415} C_VEL
LIN {X 0,Y 129.543,Z 285.549,A -85,B 0,C 180,E1 -29143.899,E2 -29143.899} C_VEL
LIN {X 0,Y 128.214,Z 281.687,A -85,B 0,C 180,E1 -29147.133,E2 -29147.133} C_VEL
LIN {X 0,Y 127.244,Z 279.05,A -85,B 0,C 180,E1 -29150.061,E2 -29150.061} C_VEL
LIN {X 0,Y 126.587,Z 277.04,A -85,B 0,C 180,E1 -29152.824,E2 -29152.824} C_VEL
LIN {X 0,Y 125.998,Z 274.074,A -85,B 0,C 180,E1 -29160,E2 -29160} C_VEL
LIN {X 0,Y 126.747,Z 277.476,A -85,B 0,C 180,E1 -29167.644,E2 -29167.644} C_VEL
LIN {X 0,Y 127.954,Z 281.002,A -85,B 0,C 180,E1 -29171.886,E2 -29171.886} C_VEL
LIN {X 0,Y 129.198,Z 284.399,A -85,B 0,C 180,E1 -29174.974,E2 -29174.974} C_VEL
LIN {X 0,Y 129.56,Z 285.571,A -85,B 0,C 180,E1 -29175.797,E2 -29175.797} C_VEL
LIN {X 0,Y 127.263,Z 299.212,A -85,B 0,C 180,E1 -29176.301,E2 -29176.301} C_VEL
LIN {X 0,Y 123.746,Z 312.054,A -85,B 0,C 180,E1 -29176.994,E2 -29176.994} C_VEL
LIN {X 0,Y 119.025,Z 324.245,A -85,B 0,C 180,E1 -29177.923,E2 -29177.923} C_VEL
LIN {X 0,Y 112.667,Z 336.809,A -85,B 0,C 180,E1 -29179.357,E2 -29179.357} C_VEL
LIN {X 0,Y 105.506,Z 347.987,A -85,B 0,C 180,E1 -29181.162,E2 -29181.162} C_VEL
LIN {X 0,Y 97.716,Z 357.91,A -85,B 0,C 180,E1 -29183.508,E2 -29183.508} C_VEL
LIN {X 0,Y 90.121,Z 366.048,A -85,B 0,C 180,E1 -29186.258,E2 -29186.258} C_VEL
LIN {X 0,Y 81.401,Z 374.041,A -85,B 0,C 180,E1 -29190.303,E2 -29190.303} C_VEL
LIN {X 0,Y 73.473,Z 380.306,A -85,B 0,C 180,E1 -29195.25,E2 -29195.25} C_VEL
LIN {X 0,Y 65.732,Z 385.536,A -85,B 0,C 180,E1 -29201.546,E2 -29201.546} C_VEL
LIN {X 0,Y 59.154,Z 389.491,A -85,B 0,C 180,E1 -29209.199,E2 -29209.199} C_VEL
LIN {X 0,Y 53.791,Z 392.416,A -85,B 0,C 180,E1 -29218.493,E2 -29218.493} C_VEL
LIN {X 0,Y 49.391,Z 394.807,A -85,B 0,C 180,E1 -29233.466,E2 -29233.466} C_VEL
LIN {X 0,Y 48.424,Z 395.417,A -85,B 0,C 180,E1 -29241.655,E2 -29241.655} C_VEL
LIN {X 0,Y 48.357,Z 395.631,A -85,B 0,C 180,E1 -29250,E2 -29250} C_VEL
LIN {X 0,Y 48.473,Z 395.397,A -85,B 0,C 180,E1 -29258.337,E2 -29258.337} C_VEL
LIN {X 0,Y 51.195,Z 393.763,A -85,B 0,C 180,E1 -29274.321,E2 -29274.321} C_VEL
LIN {X 0,Y 53.791,Z 392.348,A -85,B 0,C 180,E1 -29281.508,E2 -29281.508} C_VEL
LIN {X 0,Y 59.154,Z 389.396,A -85,B 0,C 180,E1 -29290.802,E2 -29290.802} C_VEL
LIN {X 0,Y 65.731,Z 385.405,A -85,B 0,C 180,E1 -29298.456,E2 -29298.456} C_VEL
LIN {X 0,Y 72.919,Z 380.497,A -85,B 0,C 180,E1 -29304.442,E2 -29304.442} C_VEL
LIN {X 0,Y 81.384,Z 373.818,A -85,B 0,C 180,E1 -29309.719,E2 -29309.719} C_VEL
LIN {X 0,Y 90.115,Z 365.778,A -85,B 0,C 180,E1 -29313.751,E2 -29313.751} C_VEL
LIN {X 0,Y 97.71,Z 357.585,A -85,B 0,C 180,E1 -29316.501,E2 -29316.501} C_VEL
LIN {X 0,Y 105.485,Z 347.592,A -85,B 0,C 180,E1 -29318.869,E2 -29318.869} C_VEL
LIN {X 0,Y 112.632,Z 336.286,A -85,B 0,C 180,E1 -29320.694,E2 -29320.694} C_VEL
LIN {X 0,Y 118.275,Z 325.207,A -85,B 0,C 180,E1 -29321.94,E2 -29321.94} C_VEL
LIN {X 0,Y 123.002,Z 313.357,A -85,B 0,C 180,E1 -29322.868,E2 -29322.868} C_VEL
LIN {X 0,Y 126.687,Z 300.538,A -85,B 0,C 180,E1 -29323.556,E2 -29323.556} C_VEL
LIN {X 0,Y 129.111,Z 286.966,A -85,B 0,C 180,E1 -29324.05,E2 -29324.05} C_VEL
LIN {X 0,Y 129.308,Z 285.357,A -85,B 0,C 180,E1 -29324.121,E2 -29324.121} C_VEL
LIN {X 0,Y 127.84,Z 281.211,A -85,B 0,C 180,E1 -29327.6,E2 -29327.6} C_VEL
LIN {X 0,Y 126.804,Z 278.366,A -85,B 0,C 180,E1 -29330.831,E2 -29330.831} C_VEL
LIN {X 0,Y 126.254,Z 276.732,A -85,B 0,C 180,E1 -29333.207,E2 -29333.207} C_VEL
LIN {X 0,Y 125.707,Z 273.586,A -85,B 0,C 180,E1 -29340.401,E2 -29340.401} C_VEL
LIN {X 0,Y 126.524,Z 277.458,A -85,B 0,C 180,E1 -29348.384,E2 -29348.384} C_VEL
LIN {X 0,Y 127.748,Z 280.942,A -85,B 0,C 180,E1 -29352.511,E2 -29352.511} C_VEL
LIN {X 0,Y 129.249,Z 285.218,A -85,B 0,C 180,E1 -29356.181,E2 -29356.181} C_VEL
LIN {X 0,Y 126.902,Z 298.702,A -85,B 0,C 180,E1 -29356.746,E2 -29356.746} C_VEL
LIN {X 0,Y 123.541,Z 310.723,A -85,B 0,C 180,E1 -29357.425,E2 -29357.425} C_VEL
LIN {X 0,Y 123.394,Z 311.16,A -85,B 0,C 180,E1 -29357.462,E2 -29357.462} C_VEL
LIN {X 0,Y 121.254,Z 316.699,A -85,B 0,C 180,E1 -29357.648,E2 -29357.648} C_VEL
LIN {X 0,Y 114.686,Z 328.857,A -85,B 0,C 180,E1 -29356.952,E2 -29356.952} C_VEL
LIN {X 0,Y 110.472,Z 335.534,A -85,B 0,C 180,E1 -29356.793,E2 -29356.793} C_VEL
LIN {X 0,Y 108.369,Z 338.806,A -85,B 0,C 180,E1 -29357.06,E2 -29357.06} C_VEL
LIN {X 0,Y 101.17,Z 349.153,A -85,B 0,C 180,E1 -29358.828,E2 -29358.828} C_VEL
LIN {X 0,Y 94.028,Z 357.682,A -85,B 0,C 180,E1 -29360.886,E2 -29360.886} C_VEL
LIN {X 0,Y 86.331,Z 365.536,A -85,B 0,C 180,E1 -29363.675,E2 -29363.675} C_VEL
LIN {X 0,Y 77.36,Z 373.207,A -85,B 0,C 180,E1 -29367.654,E2 -29367.654} C_VEL
LIN {X 0,Y 67.403,Z 380.258,A -85,B 0,C 180,E1 -29373.473,E2 -29373.473} C_VEL
LIN {X 0,Y 59.515,Z 384.95,A -85,B 0,C 180,E1 -29379.864,E2 -29379.864} C_VEL
LIN {X 0,Y 52.627,Z 388.534,A -85,B 0,C 180,E1 -29388.108,E2 -29388.108} C_VEL
LIN {X 0,Y 48.724,Z 390.383,A -85,B 0,C 180,E1 -29394.763,E2 -29394.763} C_VEL
LIN {X 0,Y 45.546,Z 391.769,A -85,B 0,C 180,E1 -29402.424,E2 -29402.424} C_VEL
LIN {X 0,Y 41.799,Z 393.358,A -85,B 0,C 180,E1 -29420.32,E2 -29420.32} C_VEL
LIN {X 0,Y 41.419,Z 393.58,A -85,B 0,C 180,E1 -29430,E2 -29430} C_VEL
LIN {X 0,Y 41.798,Z 393.384,A -85,B 0,C 180,E1 -29439.679,E2 -29439.679} C_VEL
LIN {X 0,Y 45.484,Z 391.829,A -85,B 0,C 180,E1 -29457.615,E2 -29457.615} C_VEL
LIN {X 0,Y 48.691,Z 390.468,A -85,B 0,C 180,E1 -29465.264,E2 -29465.264} C_VEL
LIN {X 0,Y 54.752,Z 387.592,A -85,B 0,C 180,E1 -29474.908,E2 -29474.908} C_VEL
LIN {X 0,Y 62.016,Z 383.69,A -85,B 0,C 180,E1 -29482.493,E2 -29482.493} C_VEL
LIN {X 0,Y 70.166,Z 378.653,A -85,B 0,C 180,E1 -29488.362,E2 -29488.362} C_VEL
LIN {X 0,Y 78.789,Z 372.31,A -85,B 0,C 180,E1 -29493.125,E2 -29493.125} C_VEL
LIN {X 0,Y 87.776,Z 364.38,A -85,B 0,C 180,E1 -29497.039,E2 -29497.039} C_VEL
LIN {X 0,Y 95.582,Z 356.288,A -85,B 0,C 180,E1 -29499.633,E2 -29499.633} C_VEL
LIN {X 0,Y 103.53,Z 346.415,A -85,B 0,C 180,E1 -29501.871,E2 -29501.871} C_VEL
LIN {X 0,Y 110.819,Z 335.284,A -85,B 0,C 180,E1 -29503.576,E2 -29503.576} C_VEL
LIN {X 0,Y 117.222,Z 322.925,A -85,B 0,C 180,E1 -29504.887,E2 -29504.887} C_VEL
LIN {X 0,Y 121.898,Z 310.999,A -85,B 0,C 180,E1 -29505.876,E2 -29505.876} C_VEL
LIN {X 0,Y 125.358,Z 298.875,A -85,B 0,C 180,E1 -29506.505,E2 -29506.505} C_VEL
LIN {X 0,Y 127.184,Z 289.591,A -85,B 0,C 180,E1 -29506.905,E2 -29506.905} C_VEL
LIN {X 0,Y 126.089,Z 285.875,A -85,B 0,C 180,E1 -29510.779,E2 -29510.779} C_VEL
LIN {X 0,Y 125.549,Z 283.877,A -85,B 0,C 180,E1 -29513.572,E2 -29513.572} C_VEL
LIN {X 0,Y 125.116,Z 281.255,A -85,B 0,C 180,E1 -29520,E2 -29520} C_VEL
LIN {X 0,Y 125.71,Z 284.407,A -85,B 0,C 180,E1 -29527.024,E2 -29527.024} C_VEL
LIN {X 0,Y 126.533,Z 287.347,A -85,B 0,C 180,E1 -29530.602,E2 -29530.602} C_VEL
LIN {X 0,Y 127.207,Z 289.577,A -85,B 0,C 180,E1 -29532.767,E2 -29532.767} C_VEL
LIN {X 0,Y 124.986,Z 301.158,A -85,B 0,C 180,E1 -29533.279,E2 -29533.279} C_VEL
LIN {X 0,Y 121.337,Z 313.415,A -85,B 0,C 180,E1 -29533.893,E2 -29533.893} C_VEL
LIN {X 0,Y 116.272,Z 325.699,A -85,B 0,C 180,E1 -29534.737,E2 -29534.737} C_VEL
LIN {X 0,Y 110.518,Z 336.651,A -85,B 0,C 180,E1 -29535.885,E2 -29535.885} C_VEL
LIN {X 0,Y 103.155,Z 347.828,A -85,B 0,C 180,E1 -29537.481,E2 -29537.481} C_VEL
LIN {X 0,Y 95.106,Z 357.75,A -85,B 0,C 180,E1 -29539.58,E2 -29539.58} C_VEL
LIN {X 0,Y 87.202,Z 365.888,A -85,B 0,C 180,E1 -29542.054,E2 -29542.054} C_VEL
LIN {X 0,Y 78.052,Z 373.88,A -85,B 0,C 180,E1 -29545.787,E2 -29545.787} C_VEL
LIN {X 0,Y 68.849,Z 380.633,A -85,B 0,C 180,E1 -29550.916,E2 -29550.916} C_VEL
LIN {X 0,Y 61.245,Z 385.374,A -85,B 0,C 180,E1 -29556.558,E2 -29556.558} C_VEL
LIN {X 0,Y 53.953,Z 389.329,A -85,B 0,C 180,E1 -29564.24,E2 -29564.24} C_VEL
LIN {X 0,Y 47.849,Z 392.253,A -85,B 0,C 180,E1 -29574.02,E2 -29574.02} C_VEL
LIN {X 0,Y 42.611,Z 394.645,A -85,B 0,C 180,E1 -29590.74,E2 -29590.74} C_VEL
LIN {X 0,Y 41.409,Z 395.255,A -85,B 0,C 180,E1 -29600.229,E2 -29600.229} C_VEL
LIN {X 0,Y 41.272,Z 395.469,A -85,B 0,C 180,E1 -29610,E2 -29610} C_VEL
LIN {X 0,Y 41.447,Z 395.234,A -85,B 0,C 180,E1 -29619.763,E2 -29619.763} C_VEL
LIN {X 0,Y 44.788,Z 393.599,A -85,B 0,C 180,E1 -29638.083,E2 -29638.083} C_VEL
LIN {X 0,Y 47.85,Z 392.184,A -85,B 0,C 180,E1 -29645.981,E2 -29645.981} C_VEL
LIN {X 0,Y 53.953,Z 389.232,A -85,B 0,C 180,E1 -29655.761,E2 -29655.761} C_VEL
LIN {X 0,Y 61.244,Z 385.242,A -85,B 0,C 180,E1 -29663.445,E2 -29663.445} C_VEL
LIN {X 0,Y 69.976,Z 379.674,A -85,B 0,C 180,E1 -29669.856,E2 -29669.856} C_VEL
LIN {X 0,Y 78.033,Z 373.653,A -85,B 0,C 180,E1 -29674.243,E2 -29674.243} C_VEL
LIN {X 0,Y 87.196,Z 365.613,A -85,B 0,C 180,E1 -29677.956,E2 -29677.956} C_VEL
LIN {X 0,Y 95.1,Z 357.42,A -85,B 0,C 180,E1 -29680.431,E2 -29680.431} C_VEL
LIN {X 0,Y 103.141,Z 347.426,A -85,B 0,C 180,E1 -29682.546,E2 -29682.546} C_VEL
LIN {X 0,Y 110.489,Z 336.12,A -85,B 0,C 180,E1 -29684.169,E2 -29684.169} C_VEL
LIN {X 0,Y 116.271,Z 325.04,A -85,B 0,C 180,E1 -29685.266,E2 -29685.266} C_VEL
LIN {X 0,Y 121.047,Z 313.329,A -85,B 0,C 180,E1 -29686.074,E2 -29686.074} C_VEL
LIN {X 0,Y 124.802,Z 300.631,A -85,B 0,C 180,E1 -29686.673,E2 -29686.673} C_VEL
LIN {X 0,Y 126.954,Z 289.44,A -85,B 0,C 180,E1 -29687.106,E2 -29687.106} C_VEL
LIN {X 0,Y 125.83,Z 285.698,A -85,B 0,C 180,E1 -29690.962,E2 -29690.962} C_VEL
LIN {X 0,Y 125.22,Z 283.557,A -85,B 0,C 180,E1 -29693.959,E2 -29693.959} C_VEL
LIN {X 0,Y 124.815,Z 280.845,A -85,B 0,C 180,E1 -29700.403,E2 -29700.403} C_VEL
LIN {X 0,Y 125.452,Z 284.289,A -85,B 0,C 180,E1 -29707.646,E2 -29707.646} C_VEL
LIN {X 0,Y 126.461,Z 287.888,A -85,B 0,C 180,E1 -29711.826,E2 -29711.826} C_VEL
LIN {X 0,Y 126.894,Z 289.382,A -85,B 0,C 180,E1 -29713.206,E2 -29713.206} C_VEL
LIN {X 0,Y 124.161,Z 302.355,A -85,B 0,C 180,E1 -29713.778,E2 -29713.778} C_VEL
LIN {X 0,Y 120.348,Z 314.418,A -85,B 0,C 180,E1 -29714.498,E2 -29714.498} C_VEL
LIN {X 0,Y 114.936,Z 327.101,A -85,B 0,C 180,E1 -29715.621,E2 -29715.621} C_VEL
LIN {X 0,Y 108.369,Z 338.806,A -85,B 0,C 180,E1 -29717.06,E2 -29717.06} C_VEL
LIN {X 0,Y 104.978,Z 343.656,A -85,B 0,C 180,E1 -29717.424,E2 -29717.424} C_VEL
LIN {X 0,Y 98.496,Z 351.194,A -85,B 0,C 180,E1 -29717.243,E2 -29717.243} C_VEL
LIN {X 0,Y 91.571,Z 358.222,A -85,B 0,C 180,E1 -29717.226,E2 -29717.226} C_VEL
LIN {X 0,Y 87.427,Z 362.219,A -85,B 0,C 180,E1 -29717.981,E2 -29717.981} C_VEL
LIN {X 0,Y 78.026,Z 370.535,A -85,B 0,C 180,E1 -29721.343,E2 -29721.343} C_VEL
LIN {X 0,Y 69.735,Z 376.617,A -85,B 0,C 180,E1 -29724.901,E2 -29724.901} C_VEL
LIN {X 0,Y 60.847,Z 382.111,A -85,B 0,C 180,E1 -29729.972,E2 -29729.972} C_VEL
LIN {X 0,Y 52.528,Z 386.421,A -85,B 0,C 180,E1 -29736.604,E2 -29736.604} C_VEL
LIN {X 0,Y 47.568,Z 388.698,A -85,B 0,C 180,E1 -29742.376,E2 -29742.376} C_VEL
LIN {X 0,Y 43.125,Z 390.546,A -85,B 0,C 180,E1 -29749.317,E2 -29749.317} C_VEL
LIN {X 0,Y 39.375,Z 391.932,A -85,B 0,C 180,E1 -29757.624,E2 -29757.624} C_VEL
LIN {X 0,Y 34.815,Z 393.521,A -85,B 0,C 180,E1 -29778.353,E2 -29778.353} C_VEL
LIN {X 0,Y 34.323,Z 393.742,A -85,B 0,C 180,E1 -29789.999,E2 -29789.999} C_VEL
LIN {X 0,Y 34.814,Z 393.546,A -85,B 0,C 180,E1 -29801.646,E2 -29801.646} C_VEL
LIN {X 0,Y 36.536,Z 392.959,A -85,B 0,C 180,E1 -29812.626,E2 -29812.626} C_VEL
LIN {X 0,Y 43.084,Z 390.629,A -85,B 0,C 180,E1 -29830.729,E2 -29830.729} C_VEL
LIN {X 0,Y 49.967,Z 387.754,A -85,B 0,C 180,E1 -29840.676,E2 -29840.676} C_VEL
LIN {X 0,Y 57.972,Z 383.851,A -85,B 0,C 180,E1 -29848.06,E2 -29848.06} C_VEL
LIN {X 0,Y 66.711,Z 378.814,A -85,B 0,C 180,E1 -29853.569,E2 -29853.569} C_VEL
LIN {X 0,Y 75.844,Z 372.47,A -85,B 0,C 180,E1 -29857.916,E2 -29857.916} C_VEL
LIN {X 0,Y 85.258,Z 364.54,A -85,B 0,C 180,E1 -29861.436,E2 -29861.436} C_VEL
LIN {X 0,Y 93.354,Z 356.447,A -85,B 0,C 180,E1 -29863.71,E2 -29863.71} C_VEL
LIN {X 0,Y 101.548,Z 346.574,A -85,B 0,C 180,E1 -29865.677,E2 -29865.677} C_VEL
LIN {X 0,Y 109.029,Z 335.441,A -85,B 0,C 180,E1 -29867.148,E2 -29867.148} C_VEL
LIN {X 0,Y 115.516,Z 323.214,A -85,B 0,C 180,E1 -29868.264,E2 -29868.264} C_VEL
LIN {X 0,Y 120.535,Z 310.616,A -85,B 0,C 180,E1 -29869.194,E2 -29869.194} C_VEL
LIN {X 0,Y 124.137,Z 297.989,A -85,B 0,C 180,E1 -29869.726,E2 -29869.726} C_VEL
LIN {X 0,Y 124.959,Z 294.088,A -85,B 0,C 180,E1 -29869.944,E2 -29869.944} C_VEL
LIN {X 0,Y 124.388,Z 290.901,A -85,B 0,C 180,E1 -29873.919,E2 -29873.919} C_VEL
LIN {X 0,Y 124.15,Z 288.404,A -85,B 0,C 180,E1 -29880,E2 -29880} C_VEL
LIN {X 0,Y 124.456,Z 291.095,A -85,B 0,C 180,E1 -29886.078,E2 -29886.078} C_VEL
LIN {X 0,Y 125.031,Z 294.156,A -85,B 0,C 180,E1 -29889.82,E2 -29889.82} C_VEL
LIN {X 0,Y 121.919,Z 306.951,A -85,B 0,C 180,E1 -29890.304,E2 -29890.304} C_VEL
LIN {X 0,Y 117.239,Z 319.833,A -85,B 0,C 180,E1 -29890.917,E2 -29890.917} C_VEL
LIN {X 0,Y 111.307,Z 332.129,A -85,B 0,C 180,E1 -29891.854,E2 -29891.854} C_VEL
LIN {X 0,Y 104.597,Z 343.029,A -85,B 0,C 180,E1 -29893.027,E2 -29893.027} C_VEL
LIN {X 0,Y 96.261,Z 353.863,A -85,B 0,C 180,E1 -29894.677,E2 -29894.677} C_VEL
LIN {X 0,Y 88.039,Z 362.668,A -85,B 0,C 180,E1 -29896.677,E2 -29896.677} C_VEL
LIN {X 0,Y 78.379,Z 371.249,A -85,B 0,C 180,E1 -29899.695,E2 -29899.695} C_VEL
LIN {X 0,Y 69.049,Z 378.121,A -85,B 0,C 180,E1 -29903.647,E2 -29903.647} C_VEL
LIN {X 0,Y 60.184,Z 383.631,A -85,B 0,C 180,E1 -29908.859,E2 -29908.859} C_VEL
LIN {X 0,Y 51.839,Z 387.949,A -85,B 0,C 180,E1 -29915.567,E2 -29915.567} C_VEL
LIN {X 0,Y 46.784,Z 390.239,A -85,B 0,C 180,E1 -29921.314,E2 -29921.314} C_VEL
LIN {X 0,Y 42.283,Z 392.091,A -85,B 0,C 180,E1 -29928.329,E2 -29928.329} C_VEL
LIN {X 0,Y 35.971,Z 394.483,A -85,B 0,C 180,E1 -29946.999,E2 -29946.999} C_VEL
LIN {X 0,Y 34.415,Z 395.092,A -85,B 0,C 180,E1 -29958.217,E2 -29958.217} C_VEL
LIN {X 0,Y 34.159,Z 395.307,A -85,B 0,C 180,E1 -29970.001,E2 -29970.001} C_VEL
LIN {X 0,Y 34.47,Z 395.072,A -85,B 0,C 180,E1 -29981.765,E2 -29981.765} C_VEL
LIN {X 0,Y 38.645,Z 393.436,A -85,B 0,C 180,E1 -30003.065,E2 -30003.065} C_VEL
LIN {X 0,Y 42.283,Z 392.02,A -85,B 0,C 180,E1 -30011.672,E2 -30011.672} C_VEL
LIN {X 0,Y 49.246,Z 389.068,A -85,B 0,C 180,E1 -30021.713,E2 -30021.713} C_VEL
LIN {X 0,Y 57.294,Z 385.078,A -85,B 0,C 180,E1 -30029.166,E2 -30029.166} C_VEL
LIN {X 0,Y 67.489,Z 378.959,A -85,B 0,C 180,E1 -30035.614,E2 -30035.614} C_VEL
LIN {X 0,Y 76.788,Z 372.253,A -85,B 0,C 180,E1 -30039.74,E2 -30039.74} C_VEL
LIN {X 0,Y 86.411,Z 363.959,A -85,B 0,C 180,E1 -30042.872,E2 -30042.872} C_VEL
LIN {X 0,Y 94.594,Z 355.446,A -85,B 0,C 180,E1 -30044.985,E2 -30044.985} C_VEL
LIN {X 0,Y 102.899,Z 344.933,A -85,B 0,C 180,E1 -30046.723,E2 -30046.723} C_VEL
LIN {X 0,Y 110.454,Z 333.093,A -85,B 0,C 180,E1 -30048.038,E2 -30048.038} C_VEL
LIN {X 0,Y 116.492,Z 320.838,A -85,B 0,C 180,E1 -30048.966,E2 -30048.966} C_VEL
LIN {X 0,Y 121.101,Z 308.492,A -85,B 0,C 180,E1 -30049.581,E2 -30049.581} C_VEL
LIN {X 0,Y 124.485,Z 295.498,A -85,B 0,C 180,E1 -30050.034,E2 -30050.034} C_VEL
LIN {X 0,Y 124.756,Z 293.855,A -85,B 0,C 180,E1 -30050.163,E2 -30050.163} C_VEL
LIN {X 0,Y 124.126,Z 290.549,A -85,B 0,C 180,E1 -30054.314,E2 -30054.314} C_VEL
LIN {X 0,Y 123.855,Z 288.02,A -85,B 0,C 180,E1 -30060,E2 -30060} C_VEL
LIN {X 0,Y 124.172,Z 291.143,A -85,B 0,C 180,E1 -30066.908,E2 -30066.908} C_VEL
LIN {X 0,Y 124.688,Z 293.844,A -85,B 0,C 180,E1 -30070.203,E2 -30070.203} C_VEL
LIN {X 0,Y 121.588,Z 306.322,A -85,B 0,C 180,E1 -30070.696,E2 -30070.696} C_VEL
LIN {X 0,Y 117.243,Z 318.487,A -85,B 0,C 180,E1 -30071.476,E2 -30071.476} C_VEL
LIN {X 0,Y 111.563,Z 330.427,A -85,B 0,C 180,E1 -30072.464,E2 -30072.464} C_VEL
LIN {X 0,Y 104.893,Z 341.445,A -85,B 0,C 180,E1 -30073.706,E2 -30073.706} C_VEL
LIN {X 0,Y 98.292,Z 350.371,A -85,B 0,C 180,E1 -30075.145,E2 -30075.145} C_VEL
LIN {X 0,Y 90.114,Z 359.531,A -85,B 0,C 180,E1 -30077.181,E2 -30077.181} C_VEL
LIN {X 0,Y 87.427,Z 362.219,A -85,B 0,C 180,E1 -30077.981,E2 -30077.981} C_VEL
LIN {X 0,Y 83.144,Z 366.072,A -85,B 0,C 180,E1 -30078.874,E2 -30078.874} C_VEL
LIN {X 0,Y 75.163,Z 371.919,A -85,B 0,C 180,E1 -30079.409,E2 -30079.409} C_VEL
LIN {X 0,Y 66.753,Z 377.121,A -85,B 0,C 180,E1 -30080.178,E2 -30080.178} C_VEL
LIN {X 0,Y 61.849,Z 379.948,A -85,B 0,C 180,E1 -30081.712,E2 -30081.712} C_VEL
LIN {X 0,Y 51.563,Z 385.277,A -85,B 0,C 180,E1 -30087.632,E2 -30087.632} C_VEL
LIN {X 0,Y 43.098,Z 388.861,A -85,B 0,C 180,E1 -30095.377,E2 -30095.377} C_VEL
LIN {X 0,Y 38.02,Z 390.709,A -85,B 0,C 180,E1 -30102.319,E2 -30102.319} C_VEL
LIN {X 0,Y 33.589,Z 392.095,A -85,B 0,C 180,E1 -30111.119,E2 -30111.119} C_VEL
LIN {X 0,Y 27.907,Z 393.683,A -85,B 0,C 180,E1 -30135.413,E2 -30135.413} C_VEL
LIN {X 0,Y 27.242,Z 393.904,A -85,B 0,C 180,E1 -30149.999,E2 -30149.999} C_VEL
LIN {X 0,Y 27.905,Z 393.708,A -85,B 0,C 180,E1 -30164.586,E2 -30164.586} C_VEL
LIN {X 0,Y 30.1,Z 393.121,A -85,B 0,C 180,E1 -30177.838,E2 -30177.838} C_VEL
LIN {X 0,Y 37.974,Z 390.791,A -85,B 0,C 180,E1 -30197.756,E2 -30197.756} C_VEL
LIN {X 0,Y 45.794,Z 387.916,A -85,B 0,C 180,E1 -30207.573,E2 -30207.573} C_VEL
LIN {X 0,Y 54.541,Z 384.013,A -85,B 0,C 180,E1 -30214.421,E2 -30214.421} C_VEL
LIN {X 0,Y 63.865,Z 378.975,A -85,B 0,C 180,E1 -30219.289,E2 -30219.289} C_VEL
LIN {X 0,Y 73.464,Z 372.631,A -85,B 0,C 180,E1 -30223.069,E2 -30223.069} C_VEL
LIN {X 0,Y 83.273,Z 364.699,A -85,B 0,C 180,E1 -30226.062,E2 -30226.062} C_VEL
LIN {X 0,Y 91.621,Z 356.606,A -85,B 0,C 180,E1 -30227.964,E2 -30227.964} C_VEL
LIN {X 0,Y 100.03,Z 346.732,A -85,B 0,C 180,E1 -30229.615,E2 -30229.615} C_VEL
LIN {X 0,Y 107.675,Z 335.598,A -85,B 0,C 180,E1 -30230.826,E2 -30230.826} C_VEL
LIN {X 0,Y 114.212,Z 323.522,A -85,B 0,C 180,E1 -30231.737,E2 -30231.737} C_VEL
LIN {X 0,Y 119.324,Z 311.027,A -85,B 0,C 180,E1 -30232.529,E2 -30232.529} C_VEL
LIN {X 0,Y 122.893,Z 298.842,A -85,B 0,C 180,E1 -30233.004,E2 -30233.004} C_VEL
LIN {X 0,Y 122.764,Z 297.266,A -85,B 0,C 180,E1 -30235.485,E2 -30235.485} C_VEL
LIN {X 0,Y 122.853,Z 295.483,A -85,B 0,C 180,E1 -30240,E2 -30240} C_VEL
LIN {X 0,Y 122.884,Z 297.843,A -85,B 0,C 180,E1 -30245.332,E2 -30245.332} C_VEL
LIN {X 0,Y 122.964,Z 298.831,A -85,B 0,C 180,E1 -30246.677,E2 -30246.677} C_VEL
LIN {X 0,Y 119.846,Z 309.869,A -85,B 0,C 180,E1 -30247.11,E2 -30247.11} C_VEL
LIN {X 0,Y 115.229,Z 321.711,A -85,B 0,C 180,E1 -30247.595,E2 -30247.595} C_VEL
LIN {X 0,Y 109.212,Z 333.48,A -85,B 0,C 180,E1 -30248.347,E2 -30248.347} C_VEL
LIN {X 0,Y 101.517,Z 345.22,A -85,B 0,C 180,E1 -30249.421,E2 -30249.421} C_VEL
LIN {X 0,Y 93.01,Z 355.641,A -85,B 0,C 180,E1 -30250.798,E2 -30250.798} C_VEL
LIN {X 0,Y 82.918,Z 365.568,A -85,B 0,C 180,E1 -30252.911,E2 -30252.911} C_VEL
LIN {X 0,Y 72.988,Z 373.558,A -85,B 0,C 180,E1 -30255.658,E2 -30255.658} C_VEL
LIN {X 0,Y 62.782,Z 380.273,A -85,B 0,C 180,E1 -30259.623,E2 -30259.623} C_VEL
LIN {X 0,Y 53.998,Z 385.052,A -85,B 0,C 180,E1 -30264.348,E2 -30264.348} C_VEL
LIN {X 0,Y 45.179,Z 389.005,A -85,B 0,C 180,E1 -30271.178,E2 -30271.178} C_VEL
LIN {X 0,Y 37.257,Z 391.929,A -85,B 0,C 180,E1 -30281.015,E2 -30281.015} C_VEL
LIN {X 0,Y 32.905,Z 393.322,A -85,B 0,C 180,E1 -30290.153,E2 -30290.153} C_VEL
LIN {X 0,Y 27.496,Z 394.93,A -85,B 0,C 180,E1 -30315.192,E2 -30315.192} C_VEL
LIN {X 0,Y 27.052,Z 395.144,A -85,B 0,C 180,E1 -30330.001,E2 -30330.001} C_VEL
LIN {X 0,Y 27.539,Z 394.909,A -85,B 0,C 180,E1 -30344.786,E2 -30344.786} C_VEL
LIN {X 0,Y 32.907,Z 393.273,A -85,B 0,C 180,E1 -30369.846,E2 -30369.846} C_VEL
LIN {X 0,Y 37.257,Z 391.857,A -85,B 0,C 180,E1 -30378.986,E2 -30378.986} C_VEL
LIN {X 0,Y 45.179,Z 388.904,A -85,B 0,C 180,E1 -30388.823,E2 -30388.823} C_VEL
LIN {X 0,Y 53.996,Z 384.915,A -85,B 0,C 180,E1 -30395.658,E2 -30395.658} C_VEL
LIN {X 0,Y 63.616,Z 379.596,A -85,B 0,C 180,E1 -30400.796,E2 -30400.796} C_VEL
LIN {X 0,Y 72.98,Z 373.324,A -85,B 0,C 180,E1 -30404.366,E2 -30404.366} C_VEL
LIN {X 0,Y 82.915,Z 365.283,A -85,B 0,C 180,E1 -30407.099,E2 -30407.099} C_VEL
LIN {X 0,Y 91.319,Z 357.089,A -85,B 0,C 180,E1 -30408.889,E2 -30408.889} C_VEL
LIN {X 0,Y 99.804,Z 347.095,A -85,B 0,C 180,E1 -30410.351,E2 -30410.351} C_VEL
LIN {X 0,Y 107.487,Z 335.786,A -85,B 0,C 180,E1 -30411.472,E2 -30411.472} C_VEL
LIN {X 0,Y 114.038,Z 323.59,A -85,B 0,C 180,E1 -30412.27,E2 -30412.27} C_VEL
LIN {X 0,Y 119,Z 311.417,A -85,B 0,C 180,E1 -30412.792,E2 -30412.792} C_VEL
LIN {X 0,Y 122.69,Z 298.658,A -85,B 0,C 180,E1 -30413.215,E2 -30413.215} C_VEL
LIN {X 0,Y 122.518,Z 296.968,A -85,B 0,C 180,E1 -30415.888,E2 -30415.888} C_VEL
LIN {X 0,Y 122.554,Z 295.22,A -85,B 0,C 180,E1 -30420.411,E2 -30420.411} C_VEL
LIN {X 0,Y 122.551,Z 297.757,A -85,B 0,C 180,E1 -30425.966,E2 -30425.966} C_VEL
LIN {X 0,Y 122.623,Z 298.539,A -85,B 0,C 180,E1 -30427.09,E2 -30427.09} C_VEL
LIN {X 0,Y 119.02,Z 310.914,A -85,B 0,C 180,E1 -30427.575,E2 -30427.575} C_VEL
LIN {X 0,Y 114.184,Z 322.867,A -85,B 0,C 180,E1 -30428.303,E2 -30428.303} C_VEL
LIN {X 0,Y 107.697,Z 335.006,A -85,B 0,C 180,E1 -30429.245,E2 -30429.245} C_VEL
LIN {X 0,Y 100.061,Z 346.28,A -85,B 0,C 180,E1 -30430.479,E2 -30430.479} C_VEL
LIN {X 0,Y 91.632,Z 356.235,A -85,B 0,C 180,E1 -30432.067,E2 -30432.067} C_VEL
LIN {X 0,Y 83.299,Z 364.387,A -85,B 0,C 180,E1 -30434.009,E2 -30434.009} C_VEL
LIN {X 0,Y 73.517,Z 372.37,A -85,B 0,C 180,E1 -30437.066,E2 -30437.066} C_VEL
LIN {X 0,Y 63.893,Z 378.777,A -85,B 0,C 180,E1 -30440.778,E2 -30440.778} C_VEL
LIN {X 0,Y 61.849,Z 379.948,A -85,B 0,C 180,E1 -30441.712,E2 -30441.712} C_VEL
LIN {X 0,Y 56.876,Z 382.564,A -85,B 0,C 180,E1 -30443.536,E2 -30443.536} C_VEL
LIN {X 0,Y 47.858,Z 386.311,A -85,B 0,C 180,E1 -30445.56,E2 -30445.56} C_VEL
LIN {X 0,Y 38.726,Z 389.363,A -85,B 0,C 180,E1 -30448.714,E2 -30448.714} C_VEL
LIN {X 0,Y 33.772,Z 390.828,A -85,B 0,C 180,E1 -30453.134,E2 -30453.134} C_VEL
LIN {X 0,Y 28.415,Z 392.258,A -85,B 0,C 180,E1 -30462.097,E2 -30462.097} C_VEL
LIN {X 0,Y 21.131,Z 393.845,A -85,B 0,C 180,E1 -30490.573,E2 -30490.573} C_VEL
LIN {X 0,Y 20.154,Z 394.066,A -85,B 0,C 180,E1 -30509.999,E2 -30509.999} C_VEL
LIN {X 0,Y 21.129,Z 393.869,A -85,B 0,C 180,E1 -30529.427,E2 -30529.427} C_VEL
LIN {X 0,Y 28.383,Z 392.314,A -85,B 0,C 180,E1 -30557.974,E2 -30557.974} C_VEL
LIN {X 0,Y 33.604,Z 390.953,A -85,B 0,C 180,E1 -30566.778,E2 -30566.778} C_VEL
LIN {X 0,Y 42.4,Z 388.078,A -85,B 0,C 180,E1 -30575.733,E2 -30575.733} C_VEL
LIN {X 0,Y 51.868,Z 384.174,A -85,B 0,C 180,E1 -30581.526,E2 -30581.526} C_VEL
LIN {X 0,Y 61.71,Z 379.136,A -85,B 0,C 180,E1 -30585.474,E2 -30585.474} C_VEL
LIN {X 0,Y 71.71,Z 372.792,A -85,B 0,C 180,E1 -30588.535,E2 -30588.535} C_VEL
LIN {X 0,Y 81.851,Z 364.859,A -85,B 0,C 180,E1 -30590.901,E2 -30590.901} C_VEL
LIN {X 0,Y 90.409,Z 356.765,A -85,B 0,C 180,E1 -30592.36,E2 -30592.36} C_VEL
LIN {X 0,Y 98.998,Z 346.891,A -85,B 0,C 180,E1 -30593.654,E2 -30593.654} C_VEL
LIN {X 0,Y 106.775,Z 335.755,A -85,B 0,C 180,E1 -30594.581,E2 -30594.581} C_VEL
LIN {X 0,Y 112.838,Z 324.84,A -85,B 0,C 180,E1 -30595.232,E2 -30595.232} C_VEL
LIN {X 0,Y 118.344,Z 311.941,A -85,B 0,C 180,E1 -30595.887,E2 -30595.887} C_VEL
LIN {X 0,Y 120.905,Z 303.954,A -85,B 0,C 180,E1 -30596.191,E2 -30596.191} C_VEL
LIN {X 0,Y 121.099,Z 302.526,A -85,B 0,C 180,E1 -30600,E2 -30600} C_VEL
LIN {X 0,Y 120.982,Z 303.886,A -85,B 0,C 180,E1 -30603.522,E2 -30603.522} C_VEL
LIN {X 0,Y 116.629,Z 316.628,A -85,B 0,C 180,E1 -30603.912,E2 -30603.912} C_VEL
LIN {X 0,Y 111.016,Z 328.649,A -85,B 0,C 180,E1 -30604.393,E2 -30604.393} C_VEL
LIN {X 0,Y 104.069,Z 340.179,A -85,B 0,C 180,E1 -30605.067,E2 -30605.067} C_VEL
LIN {X 0,Y 96.266,Z 350.564,A -85,B 0,C 180,E1 -30605.904,E2 -30605.904} C_VEL
LIN {X 0,Y 88.499,Z 359.056,A -85,B 0,C 180,E1 -30606.948,E2 -30606.948} C_VEL
LIN {X 0,Y 78.2,Z 368.26,A -85,B 0,C 180,E1 -30608.666,E2 -30608.666} C_VEL
LIN {X 0,Y 68.018,Z 375.667,A -85,B 0,C 180,E1 -30611.012,E2 -30611.012} C_VEL
LIN {X 0,Y 58.017,Z 381.62,A -85,B 0,C 180,E1 -30614.282,E2 -30614.282} C_VEL
LIN {X 0,Y 48.231,Z 386.321,A -85,B 0,C 180,E1 -30618.714,E2 -30618.714} C_VEL
LIN {X 0,Y 38.871,Z 389.915,A -85,B 0,C 180,E1 -30625.311,E2 -30625.311} C_VEL
LIN {X 0,Y 33.017,Z 391.766,A -85,B 0,C 180,E1 -30631.631,E2 -30631.631} C_VEL
LIN {X 0,Y 23.515,Z 394.158,A -85,B 0,C 180,E1 -30653.292,E2 -30653.292} C_VEL
LIN {X 0,Y 20.692,Z 394.768,A -85,B 0,C 180,E1 -30670.145,E2 -30670.145} C_VEL
LIN {X 0,Y 19.959,Z 394.982,A -85,B 0,C 180,E1 -30690.001,E2 -30690.001} C_VEL
LIN {X 0,Y 20.747,Z 394.747,A -85,B 0,C 180,E1 -30709.801,E2 -30709.801} C_VEL
LIN {X 0,Y 27.807,Z 393.109,A -85,B 0,C 180,E1 -30739.309,E2 -30739.309} C_VEL
LIN {X 0,Y 33.017,Z 391.693,A -85,B 0,C 180,E1 -30748.369,E2 -30748.369} C_VEL
LIN {X 0,Y 41.936,Z 388.741,A -85,B 0,C 180,E1 -30757.182,E2 -30757.182} C_VEL
LIN {X 0,Y 51.473,Z 384.751,A -85,B 0,C 180,E1 -30762.893,E2 -30762.893} C_VEL
LIN {X 0,Y 62.814,Z 378.716,A -85,B 0,C 180,E1 -30767.476,E2 -30767.476} C_VEL
LIN {X 0,Y 73.088,Z 371.923,A -85,B 0,C 180,E1 -30770.274,E2 -30770.274} C_VEL
LIN {X 0,Y 83.335,Z 363.629,A -85,B 0,C 180,E1 -30772.275,E2 -30772.275} C_VEL
LIN {X 0,Y 91.939,Z 355.115,A -85,B 0,C 180,E1 -30773.587,E2 -30773.587} C_VEL
LIN {X 0,Y 100.594,Z 344.601,A -85,B 0,C 180,E1 -30774.61,E2 -30774.61} C_VEL
LIN {X 0,Y 107.536,Z 334.193,A -85,B 0,C 180,E1 -30775.313,E2 -30775.313} C_VEL
LIN {X 0,Y 113.648,Z 322.705,A -85,B 0,C 180,E1 -30775.875,E2 -30775.875} C_VEL
LIN {X 0,Y 118.463,Z 310.814,A -85,B 0,C 180,E1 -30776.222,E2 -30776.222} C_VEL
LIN {X 0,Y 120.688,Z 303.709,A -85,B 0,C 180,E1 -30776.451,E2 -30776.451} C_VEL
LIN {X 0,Y 120.817,Z 302.267,A -85,B 0,C 180,E1 -30780.417,E2 -30780.417} C_VEL
LIN {X 0,Y 120.618,Z 303.736,A -85,B 0,C 180,E1 -30783.898,E2 -30783.898} C_VEL
